    GVL.g_stTrackingQueue_B.Objects[2].Valid := TRUE;
    GVL.g_stTrackingQueue_B.Objects[2].ObjectID :=
        GVL.g_stTrackingQueue_B.NextObjectID;
    GVL.g_stTrackingQueue_B.Objects[2].ProductClassID := 1;
    GVL.g_stTrackingQueue_B.Objects[2].Reserved := FALSE;
    GVL.g_stTrackingQueue_B.Objects[2].ReservedToolID := 0;
    GVL.g_stTrackingQueue_B.Objects[2].CanPick := TRUE;
    GVL.g_stTrackingQueue_B.Objects[2].OrientationValid := TRUE;
    GVL.g_stTrackingQueue_B.Objects[2].VisionScore := 100.0;
    GVL.g_stTrackingQueue_B.Objects[2].State := E_TrackingObjectState.OBJ_READY;

    // Đặt cách Object 1 một khoảng để dễ quan sát.
    GVL.g_stTrackingQueue_B.Objects[2].VisionPos.X := 260.0;
    GVL.g_stTrackingQueue_B.Objects[2].VisionPos.Y := 0.0;
    GVL.g_stTrackingQueue_B.Objects[2].VisionPos.Z := 50.0;
    GVL.g_stTrackingQueue_B.Objects[2].VisionPos.A := 0.0;
	
	//-------------------------------------------------------------------------
	// OBJECT 2 - POSE CHUẨN TRONG HỆ CONVEYOR
	//-------------------------------------------------------------------------
	GVL.g_stTrackingQueue_B.Objects[2].PoseInConveyor.X := 260.0;
	GVL.g_stTrackingQueue_B.Objects[2].PoseInConveyor.Y := 0.0;
	GVL.g_stTrackingQueue_B.Objects[2].PoseInConveyor.Z := 50.0;
	GVL.g_stTrackingQueue_B.Objects[2].PoseInConveyor.A := 0.0;

	
	GVL.g_stTrackingQueue_B.Objects[2].CaptureConveyorPositionMM :=
		REAL_TO_LREAL(GVL.g_aConveyorRuntime[2].Status.PositionMM);

    GVL.g_stTrackingQueue_B.ValidCount := 2;
    GVL.g_stTrackingQueue_B.ActiveIndex := GVL.C_INVALID_INDEX;
	

//     GVL.g_stTrackingQueue_B.ValidCount := 1;
    GVL.g_stTrackingQueue_B.ActiveIndex := GVL.C_INVALID_INDEX;
END_IF;


//=============================================================================
// KHỞI TẠO CẤU HÌNH MẶC ĐỊNH CHO MULTI-TOOL ROBOT B
//-----------------------------------------------------------------------------
// Chỉ chạy một lần khi cấu hình chưa được khởi tạo hoặc khi người dùng yêu cầu
// khởi tạo lại. Không ghi đè cấu hình HMI trong mỗi vòng quét PLC.
//=============================================================================
IF (NOT GVL.g_xMultiToolConfigInitializedB OR GVL.g_xInitializeMultiToolConfigB) AND (1=2) THEN

    //-------------------------------------------------------------------------
    // TOOL 1
    //-------------------------------------------------------------------------
	GVL.g_aToolConfigB[1].Enable := TRUE;
	GVL.g_aToolConfigB[1].AllowTracking := TRUE;
	GVL.g_aToolConfigB[1].ToolID := 1;
	GVL.g_aToolConfigB[1].AllowedProductClassID := 0;
	

    //-------------------------------------------------------------------------
    // RECIPE 1 DÙNG CHO COMMISSIONING
    //-------------------------------------------------------------------------
    GVL.g_aMultiTrackRecipeB[1].Enable := TRUE;
    GVL.g_aMultiTrackRecipeB[1].RecipeID := 1;
    GVL.g_aMultiTrackRecipeB[1].ProductClassID := 0;
    GVL.g_aMultiTrackRecipeB[1].TargetPickCount := 1;
    GVL.g_aMultiTrackRecipeB[1].ToolEnableMask := DWORD#1;
	
	GVL.g_aToolConfigB[1].PickOffset.X := 0.0;
	GVL.g_aToolConfigB[1].PickOffset.Y := 0.0;
	GVL.g_aToolConfigB[1].PickOffset.Z := 50.0;
	GVL.g_aToolConfigB[1].PickOffset.A := 0.0;
	
	GVL.g_aToolConfigB[1].ApproachHeight := 20.0;
	GVL.g_aToolConfigB[1].UseUpDown := FALSE;
	GVL.g_aToolConfigB[1].UpDownStroke := 20.0;
	
	GVL.g_stTrackingConfig_B.RetractHeight := 20.0;
	
	
	//-------------------------------------------------------------------------
	// TOOL 2
	//-------------------------------------------------------------------------
	GVL.g_aToolConfigB[2].Enable := TRUE;
	GVL.g_aToolConfigB[2].AllowTracking := TRUE;
	GVL.g_aToolConfigB[2].ToolID := 2;
	GVL.g_aToolConfigB[2].AllowedProductClassID := 0;
	
	GVL.g_aToolConfigB[2].PickOffset.X := 0.0;
	GVL.g_aToolConfigB[2].PickOffset.Y := 0.0;
	GVL.g_aToolConfigB[2].PickOffset.Z := 50.0;
	GVL.g_aToolConfigB[2].PickOffset.A := 0.0;
	
	GVL.g_aToolConfigB[2].ApproachHeight := 20.0;
	
	// Có thể đặt khác Tool 1 để quan sát.
	GVL.g_aToolConfigB[2].UseUpDown := FALSE;
	GVL.g_aToolConfigB[2].UpDownStroke := 20.0;
	
	GVL.g_aToolConfigB[2].Priority := 2;


	//=============================================================================
	// DYNAMIC APPROACH
	//-----------------------------------------------------------------------------
	// Thông số thử nghiệm ban đầu. Có thể chỉnh lại trên HMI sau.
	//=============================================================================
	GVL.g_stTrackingConfig_B.Motion.Approach.Speed := 100.0;
	GVL.g_stTrackingConfig_B.Motion.Approach.Acceleration := 500.0;
	GVL.g_stTrackingConfig_B.Motion.Approach.Deceleration := 500.0;
	GVL.g_stTrackingConfig_B.Motion.Approach.Jerk := 1000.0;
	GVL.g_stTrackingConfig_B.Motion.Approach.BlendRadius := 0.0;
	
	GVL.g_stTrackingSimulation.VirtualEncoderStepPerCycle := -5;

    //-------------------------------------------------------------------------
    // ĐÁNH DẤU ĐÃ KHỞI TẠO
    //-------------------------------------------------------------------------
    GVL.g_xMultiToolConfigInitializedB := TRUE;
    GVL.g_xInitializeMultiToolConfigB := FALSE;

END_IF;

//=============================================================================
// PHỤC HỒI DỮ LIỆU COMMISSIONING KHI RESET MULTI-TOOL
//-----------------------------------------------------------------------------
// Chỉ dùng khi test Object cố định.
// Khi chạy Vision/Sensor thật, Object lỗi phải được loại bỏ hoặc nạp Object mới.
//=============================================================================
IF GVL.g_xMultiTrackResetTestB THEN


	//---------------------------------------------------------------------
    // RESET TOOL 1
    //---------------------------------------------------------------------
    GVL.g_aToolStatusB[1].Busy := FALSE;
    GVL.g_aToolStatusB[1].Occupied := FALSE;
    GVL.g_aToolStatusB[1].Error := FALSE;
    GVL.g_aToolStatusB[1].ErrorID := 0;
    GVL.g_aToolStatusB[1].HeldObjectID := 0;
    GVL.g_aToolStatusB[1].GripOK := FALSE;

    //---------------------------------------------------------------------
    // RESET TOOL 2
    //---------------------------------------------------------------------
    GVL.g_aToolStatusB[2].Busy := FALSE;
    GVL.g_aToolStatusB[2].Occupied := FALSE;
    GVL.g_aToolStatusB[2].Error := FALSE;
    GVL.g_aToolStatusB[2].ErrorID := 0;
    GVL.g_aToolStatusB[2].HeldObjectID := 0;
    GVL.g_aToolStatusB[2].GripOK := FALSE;
	
	// Comment lai vi dang test object thuc

//     //---------------------------------------------------------------------
//     // RESET OBJECT 1
//     //---------------------------------------------------------------------
//     GVL.g_stTrackingQueue_B.Objects[1].Valid := TRUE;
//     GVL.g_stTrackingQueue_B.Objects[1].CanPick := TRUE;
//     GVL.g_stTrackingQueue_B.Objects[1].Reserved := FALSE;
//     GVL.g_stTrackingQueue_B.Objects[1].ReservedToolID := 0;
//     GVL.g_stTrackingQueue_B.Objects[1].State :=
//         E_TrackingObjectState.OBJ_READY;
// 
//     //---------------------------------------------------------------------
//     // RESET OBJECT 2
//     //---------------------------------------------------------------------
//     GVL.g_stTrackingQueue_B.Objects[2].Valid := TRUE;
//     GVL.g_stTrackingQueue_B.Objects[2].CanPick := TRUE;
//     GVL.g_stTrackingQueue_B.Objects[2].Reserved := FALSE;
//     GVL.g_stTrackingQueue_B.Objects[2].ReservedToolID := 0;
//     GVL.g_stTrackingQueue_B.Objects[2].State :=
//         E_TrackingObjectState.OBJ_READY;
// 
//     GVL.g_stTrackingQueue_B.ValidCount := 2;
//     GVL.g_stTrackingQueue_B.ActiveIndex := GVL.C_INVALID_INDEX;

END_IF;

IF stCommandB.Reset THEN
    udiDebugCoreStartCountB := 0;
    udiDebugExecuteToCoreCountB := 0;
    udiDebugCoreRequestCountB := 0;

    xDebugCoreStartLatchedB := FALSE;
    xDebugExecuteToCoreLatchedB := FALSE;
    xDebugCoreRequestLatchedB := FALSE;
	GVL.g_xMultiTrackStartTestB := FALSE;
END_IF;

//=============================================================================
// 04. MULTI-TOOL CONTROLLER
//-----------------------------------------------------------------------------
// Controller đọc phản hồi của Core, SelectTool và ToolManager từ vòng quét trước.
//=============================================================================
fbControllerB(
    Command := stCommandB,
    CoreAccepted := fbCoreInterfaceB.Accepted,
    CoreBusy := fbCoreInterfaceB.Busy,
    CoreSyncOK := fbCoreInterfaceB.SyncOK,
    CorePCSInUse := fbCoreInterfaceB.PCSInUse,
    CoreReleased := fbCoreInterfaceB.Released,
    CoreError := fbCoreInterfaceB.Error,
    CoreErrorID := fbCoreInterfaceB.ErrorID,
    SelectToolDone := fbSelectToolB.Done,
    SelectToolError := fbSelectToolB.Error,
    SelectToolErrorID := fbSelectToolB.ErrorID,
    Queue := GVL.g_stTrackingQueue_B,
    ToolConfig := GVL.g_aToolConfigB,
    ToolStatus := GVL.g_aToolStatusB,
    Recipes := GVL.g_aMultiTrackRecipeB,
    Status := GVL.g_stMultiTrackStatusB
);


//=============================================================================
// MULTI-TOOL TRACKING RESULT LATCH
//=============================================================================

// Command mới được Controller nhận -> xóa kết quả command trước.
IF GVL.g_stMultiTrackStatusB.Accepted THEN
    GVL.g_xTrackOKB := FALSE;
    GVL.g_xTrackErrorB := FALSE;
    GVL.g_udiTrackErrorIDB := 0;
END_IF;


//-----------------------------------------------------------------------------
// TRACKING PICK HOÀN THÀNH ĐỦ SỐ LƯỢNG.
//-----------------------------------------------------------------------------
IF GVL.g_stMultiTrackStatusB.Done
AND NOT GVL.g_stMultiTrackStatusB.Error
AND GVL.g_stMultiTrackStatusB.PickedCount >= GVL.g_stMultiTrackStatusB.TargetPickCount THEN

    GVL.g_xTrackOKB := TRUE;
    GVL.g_xTrackErrorB := FALSE;
    GVL.g_udiTrackErrorIDB := 0;

    // Chốt CommandID của đúng lệnh vừa hoàn thành.
    GVL.g_udiTrackDoneCommandIDB :=
        GVL.g_stMultiTrackStatusB.ResponseCommandID;

END_IF;


//-----------------------------------------------------------------------------
// TRACKING ERROR.
//-----------------------------------------------------------------------------
IF GVL.g_stMultiTrackStatusB.Error THEN

    GVL.g_xTrackOKB := FALSE;
    GVL.g_xTrackErrorB := TRUE;
    GVL.g_udiTrackErrorIDB :=
        GVL.g_stMultiTrackStatusB.ErrorID;

END_IF;


//-----------------------------------------------------------------------------
// RESET.
//-----------------------------------------------------------------------------
IF stCommandB.Reset THEN

    GVL.g_xTrackOKB := FALSE;
    GVL.g_xTrackErrorB := FALSE;
    GVL.g_udiTrackErrorIDB := 0;
    GVL.g_udiTrackDoneCommandIDB := 0;

END_IF;



//=============================================================================
// 05. TRACKING CORE INTERFACE
//-----------------------------------------------------------------------------
// Interface giữ Execute cho Tracking Core và chỉ hạ sau khi PCS đã release.
//=============================================================================
fbCoreInterfaceB(
    Enable := TRUE,
    Reset := fbControllerB.CoreReset,
    Abort := fbControllerB.CoreAbort,
    StartTracking := fbControllerB.CoreStart,
    ReleaseTracking := fbControllerB.CoreRelease,
    ObjectIndex := fbControllerB.CoreObjectIndex,
    ToolID := fbControllerB.CoreToolID,
    PickOffset := fbControllerB.CorePickOffset,
    ApproachHeight := fbControllerB.CoreApproachHeight,
	PickSurfaceHeightMM := fbControllerB.CorePickSurfaceHeightMM,
    CoreAccepted := GVL.g_stTrackingRuntime_B.Response.Accepted,
	CoreBusy := GVL.g_stTrackingRuntime_B.Response.Busy,
	CoreSyncOK := fbTrackingManagerB.SyncOK,
	CorePCSInUse := GVL.g_stTrackingRuntime_B.PCSInfo.InUse,
	CoreReleased := fbTrackingManagerB.Released,
	CoreError := GVL.g_stTrackingRuntime_B.Response.Error,
	CoreErrorID := GVL.g_stTrackingRuntime_B.Response.ErrorID,
	UseUpDown := fbControllerB.CoreUseUpDown,
	UpDownStroke := fbControllerB.CoreUpDownStroke,
);


//=============================================================================
// 06. CHỌN TOOL/TCP ROBOT B
//-----------------------------------------------------------------------------
// FB_SelectRobotTool phải gọi SMC_GroupSetTool thực tế, không dùng placeholder.
//=============================================================================
fbSelectToolB(
    Execute := fbControllerB.SelectToolExecute,
    Reset := stCommandB.Reset,
    ToolID := fbControllerB.SelectToolID
);


// xTrackingRequestValid :=
//     fbCoreInterfaceB.ExecuteToCore
//     AND fbCoreInterfaceB.ActiveObjectIndex >= 1
//     AND fbCoreInterfaceB.ActiveObjectIndex <= GVL.C_MAX_TRACK_OBJECTS
//     AND GVL.g_stTrackingQueue_B.Objects[fbCoreInterfaceB.ActiveObjectIndex].Valid;
	
xCoreRequestValid := fbCoreInterfaceB.ExecuteToCore
AND fbCoreInterfaceB.ActiveObjectIndex >= 1
AND fbCoreInterfaceB.ActiveObjectIndex <= GVL.C_MAX_TRACK_OBJECTS
AND GVL.g_stTrackingQueue_B.Objects[fbCoreInterfaceB.ActiveObjectIndex].Valid;

rtDebugCoreStartB(CLK := fbControllerB.CoreStart);
rtDebugExecuteToCoreB(CLK := fbCoreInterfaceB.ExecuteToCore);
rtDebugCoreRequestValidB(CLK := xCoreRequestValid);

IF rtDebugCoreStartB.Q THEN
    udiDebugCoreStartCountB := udiDebugCoreStartCountB + 1;
    xDebugCoreStartLatchedB := TRUE;
END_IF;

IF rtDebugExecuteToCoreB.Q THEN
    udiDebugExecuteToCoreCountB := udiDebugExecuteToCoreCountB + 1;
    xDebugExecuteToCoreLatchedB := TRUE;
END_IF;

IF rtDebugCoreRequestValidB.Q THEN
    udiDebugCoreRequestCountB := udiDebugCoreRequestCountB + 1;
    xDebugCoreRequestLatchedB := TRUE;
END_IF;


//=============================================================================
// 07. TRACKING CORE
//-----------------------------------------------------------------------------
// Multi-tool mode luôn dùng UseExternalSelection = TRUE.
// Controller đã chọn ObjectIndex và PickOffset theo Tool.
//=============================================================================
fbTrackingManagerB(
    Execute := xCoreRequestValid,
    Reset := fbCoreInterfaceB.ResetToCore OR stCommandB.Reset,
    Config := GVL.g_stTrackingConfig_B,
    ConveyorConfig := GVL.g_aConveyorRuntime[2].Config,
    ConveyorStatus := GVL.g_aConveyorRuntime[2].Status,
    ConveyorOrigin := stConveyorOriginB,
    VacuumOK := FALSE,
    MotionAccepted := GVL.g_xTrackingMotionAcceptedB,
    MotionBusy := GVL.g_xTrackingMotionBusyB,
    MotionDone := GVL.g_xTrackingMotionDoneB,
    MotionError := GVL.g_xTrackingMotionErrorB,
    MotionErrorID := GVL.g_udiTrackingMotionErrorIDB,
    MotionAbortDone := GVL.g_xTrackingMotionAbortDoneB,
    TestFixedObjectMode := FALSE,
    FixedObjectPosition := stFixedObjectPositionB,
    UseExternalSelection := TRUE,
    ExternalObjectIndex := fbCoreInterfaceB.ActiveObjectIndex,
    ExternalPickOffset := fbCoreInterfaceB.ActivePickOffset,
    ExternalApproachHeight := fbCoreInterfaceB.ActiveApproachHeight,
    PickerSafe := fbCoreInterfaceB.PickerSafeToCore,
    Queue := GVL.g_stTrackingQueue_B,
    Runtime := GVL.g_stTrackingRuntime_B,
	ExternalUseUpDown := fbCoreInterfaceB.ActiveUseUpDown,
	ExternalUpDownStroke := fbCoreInterfaceB.ActiveUpDownStroke,
	ExternalPickSurfaceHeightMM := fbCoreInterfaceB.ActivePickSurfaceHeightMM,
);


//=============================================================================
// 08. MAP PHẢN HỒI TRACKING CORE
//-----------------------------------------------------------------------------
// Các biến này được FB_TrackingCoreInterface_A đọc ở vòng quét tiếp theo.
//=============================================================================
GVL.g_xTrackingCoreAcceptedB := GVL.g_stTrackingRuntime_B.Response.Accepted;
GVL.g_xTrackingCoreBusyB := GVL.g_stTrackingRuntime_B.Response.Busy;
GVL.g_xTrackingCoreSyncOKB := fbTrackingManagerB.SyncOK;
GVL.g_xTrackingCorePCSInUseB := GVL.g_stTrackingRuntime_B.PCSInfo.InUse;
GVL.g_xTrackingCoreReleasedB := fbTrackingManagerB.Released;
GVL.g_xTrackingCoreErrorB := GVL.g_stTrackingRuntime_B.Response.Error;
GVL.g_udiTrackingCoreErrorIDB := GVL.g_stTrackingRuntime_B.Response.ErrorID;


//=============================================================================
// 09. MOTION QUEUE ADAPTER
//-----------------------------------------------------------------------------
// Chỉ instance này được đưa motion Tracking vào Motion Queue Robot B.
//=============================================================================
fbMotionAdapterB(
    Enable := TRUE,
    Reset := fbCoreInterfaceB.ResetToCore OR stCommandB.Reset,
    Request := fbTrackingManagerB.MotionRequest,
    Abort := fbTrackingManagerB.MotionAbort,
    Target := fbTrackingManagerB.MotionTarget,
    Speed := fbTrackingManagerB.MotionSpeed,
    Acceleration := fbTrackingManagerB.MotionAcceleration,
    Deceleration := fbTrackingManagerB.MotionDeceleration,
    Jerk := fbTrackingManagerB.MotionJerk,
    BlendRadius := fbTrackingManagerB.MotionBlendRadius,
    CoordSystem := fbTrackingManagerB.MotionCoordSystem,
    Command := fbTrackingManagerB.MotionCommand,
    LogicSimulation := GVL.g_stTrackingSimulation.Mode = E_ApplicationSimulationMode.SIM_LOGIC_ONLY,
    LogicMotionDuration := GVL.g_stTrackingSimulation.LogicMotionDuration,
    Accepted => GVL.g_xTrackingMotionAcceptedB,
    Busy => GVL.g_xTrackingMotionBusyB,
    Done => GVL.g_xTrackingMotionDoneB,
    Error => GVL.g_xTrackingMotionErrorB,
    ErrorID => GVL.g_udiTrackingMotionErrorIDB,
    AbortDone => GVL.g_xTrackingMotionAbortDoneB
);


//=============================================================================
// 10. PHÂN PHỐI COMMAND TỚI TỪNG TOOL MANAGER
//-----------------------------------------------------------------------------
// Chỉ Tool có ToolID trùng Command mới nhận Execute.
// Các Tool còn lại vẫn được gọi mỗi vòng quét để duy trì Runtime và Output.
//=============================================================================
FOR uiTool := 1 TO GVL.C_MAX_TOOLS DO
	
	// Tất cả OUTPUT mặc định Active HIGH.
	GVL.g_aToolConfigB[uiTool].IO.DownDOActiveLevel := TRUE;
	GVL.g_aToolConfigB[uiTool].IO.UpDOActiveLevel := TRUE;
	GVL.g_aToolConfigB[uiTool].IO.GripDOActiveLevel := TRUE;
	GVL.g_aToolConfigB[uiTool].IO.ReleaseDOActiveLevel := TRUE;
	
	// Tất cả INPUT feedback mặc định Active HIGH.
	GVL.g_aToolConfigB[uiTool].IO.DownOKDIActiveLevel := TRUE;
	GVL.g_aToolConfigB[uiTool].IO.UpOKDIActiveLevel := TRUE;
	GVL.g_aToolConfigB[uiTool].IO.GripOKDIActiveLevel := TRUE;
	GVL.g_aToolConfigB[uiTool].IO.PartPresentDIActiveLevel := TRUE;
	
    astToolCommandB[uiTool].Execute := FALSE;
    astToolCommandB[uiTool].Reset := stCommandB.Reset;
    astToolCommandB[uiTool].Abort := stCommandB.Abort;
    astToolCommandB[uiTool].CommandID := 0;
    astToolCommandB[uiTool].ToolID := GVL.g_aToolConfigB[uiTool].ToolID;
    astToolCommandB[uiTool].CommandType := E_ToolCommandType.NONE;
    astToolCommandB[uiTool].ObjectID := 0;

    //IF fbControllerB.ToolCommand.ToolID = GVL.g_aToolConfigB[uiTool].ToolID THEN astToolCommandB[uiTool] := fbControllerB.ToolCommand; END_IF;
	
//-------------------------------------------------------------------------
	// ƯU TIÊN 1: Command từ MultiTool Tracking Controller.
	//-------------------------------------------------------------------------
	IF fbControllerB.ToolCommand.Execute
	AND fbControllerB.ToolCommand.ToolID = GVL.g_aToolConfigB[uiTool].ToolID THEN
	
		astToolCommandB[uiTool] := fbControllerB.ToolCommand;
	
	
	//-------------------------------------------------------------------------
	// ƯU TIÊN 2: Command Tool độc lập từ Interpreter.
	// Chỉ chạy khi Controller không phát Tool Command.
	//-------------------------------------------------------------------------
	ELSIF GVL.g_stInterpreterToolCommandB.Execute
	AND GVL.g_stInterpreterToolCommandB.ToolID = GVL.g_aToolConfigB[uiTool].ToolID THEN
	
		astToolCommandB[uiTool] :=
			GVL.g_stInterpreterToolCommandB;
	
	END_IF;

    fbToolManagerB[uiTool](
        Enable := GVL.g_aToolConfigB[uiTool].Enable,
        Command := astToolCommandB[uiTool],
        Config := GVL.g_aToolConfigB[uiTool],
        Status := GVL.g_aToolStatusB[uiTool]
    );
END_FOR;


//=============================================================================
// 11. BIẾN GIÁM SÁT HMI / DEBUG
//=============================================================================
GVL.g_xMultiTrackCoreExecuteB := fbCoreInterfaceB.ExecuteToCore;
GVL.g_xMultiTrackCoreResetB := fbCoreInterfaceB.ResetToCore;
GVL.g_xMultiTrackCoreAbortB := fbCoreInterfaceB.AbortToCore;
GVL.g_xMultiTrackPickerSafeB := fbCoreInterfaceB.PickerSafeToCore;
GVL.g_uiMultiTrackObjectIndexB := fbCoreInterfaceB.ActiveObjectIndex;
GVL.g_uiMultiTrackToolIDB := fbCoreInterfaceB.ActiveToolID;
GVL.g_stMultiTrackPickOffsetB := fbCoreInterfaceB.ActivePickOffset;
GVL.g_rMultiTrackApproachHeightB := fbCoreInterfaceB.ActiveApproachHeight;
GVL.g_xSelectToolExecuteB := fbControllerB.SelectToolExecute;
GVL.g_uiSelectToolIDB := fbControllerB.SelectToolID;
GVL.g_stSelectToolTCPB := fbControllerB.SelectToolTCP;
GVL.g_xSelectToolDoneB := fbSelectToolB.Done;
GVL.g_xSelectToolErrorB := fbSelectToolB.Error;
GVL.g_udiSelectToolErrorIDB := fbSelectToolB.ErrorID;


//=============================================================================
// 12. OUTPUT CŨ CỦA TRACKING CORE
//-----------------------------------------------------------------------------
// Multi-tool mode không dùng VacuumCommand/BlowCommand; giữ map để debug.
//=============================================================================
GVL.g_xTrackingVacuumOutputB := fbTrackingManagerB.VacuumCommand;
GVL.g_xTrackingBlowOutputB := fbTrackingManagerB.BlowCommand;

END_PROGRAM

// Just_Motion_Control_x86_64_Linux_SM_WV/Application/FB_/ConveyorTrack/FB_MultiToolTrackingController_B
FUNCTION_BLOCK FB_MultiToolTrackingController_B
VAR_INPUT
    Command : ST_MultiToolTrackingCommand; // Biến nội bộ Command.
    CoreAccepted : BOOL; // Biến nội bộ CoreAccepted.
    CoreBusy : BOOL; // Biến nội bộ CoreBusy.
    CoreSyncOK : BOOL; // Biến nội bộ CoreSyncOK.
    CorePCSInUse : BOOL; // Biến nội bộ CorePCSInUse.
    CoreReleased : BOOL; // Biến nội bộ CoreReleased.
    CoreError : BOOL; // Biến nội bộ CoreError.
    CoreErrorID : UDINT; // Biến nội bộ CoreErrorID.
    SelectToolDone : BOOL; // Biến nội bộ SelectToolDone.
    SelectToolError : BOOL; // Biến nội bộ SelectToolError.
    SelectToolErrorID : UDINT; // Biến nội bộ SelectToolErrorID.
END_VAR

VAR_IN_OUT
    Queue : ST_TRACKING_QUEUE; // Biến nội bộ Queue.
    ToolConfig : ARRAY[0..GVL.C_MAX_TOOLS] OF ST_ToolConfig; // Biến nội bộ ToolConfig.
    ToolStatus : ARRAY[0..GVL.C_MAX_TOOLS] OF ST_ToolStatus; // Biến nội bộ ToolStatus.
    Recipes : ARRAY[0..GVL.C_MAX_TRACK_RECIPES] OF ST_MultiToolTrackingRecipe; // Biến nội bộ Recipes.
    Status : ST_MultiToolTrackingStatus; // Biến nội bộ Status.
END_VAR

VAR_OUTPUT
    CoreStart : BOOL; // Biến nội bộ CoreStart.
    CoreRelease : BOOL; // Biến nội bộ CoreRelease.
    CoreAbort : BOOL; // Biến nội bộ CoreAbort.
    CoreReset : BOOL; // Biến nội bộ CoreReset.
    CoreObjectIndex : UINT; // Biến nội bộ CoreObjectIndex.
    CoreToolID : UINT; // Biến nội bộ CoreToolID.
    CorePickOffset : ST_POS; // Biến nội bộ CorePickOffset.
    CoreApproachHeight : REAL; // Biến nội bộ CoreApproachHeight.
    ToolCommand : ST_ToolCommand; // Biến nội bộ ToolCommand.
    SelectToolExecute : BOOL; // Biến nội bộ SelectToolExecute.
    SelectToolID : UINT; // Biến nội bộ SelectToolID.
    SelectToolTCP : ST_POS; // Biến nội bộ SelectToolTCP.
    CoreUseUpDown : BOOL; // Biến nội bộ CoreUseUpDown.
    CoreUpDownStroke : REAL; // Biến nội bộ CoreUpDownStroke.
    CorePickSurfaceHeightMM : REAL; // Biến nội bộ CorePickSurfaceHeightMM.
END_VAR

VAR
    rtExecute : R_TRIG; // Biến nội bộ rtExecute.
    fbScheduler : FB_ToolObjectScheduler; // Biến nội bộ fbScheduler.
    stRecipe : ST_MultiToolTrackingRecipe; // Biến nội bộ stRecipe.
    uiToolIndex : UINT; // Biến nội bộ uiToolIndex.
    uiObjectIndex : UINT; // Biến nội bộ uiObjectIndex.
    uiTargetCount : UINT; // Biến nội bộ uiTargetCount.
    dwToolMask : DWORD; // Biến nội bộ dwToolMask.
    udiToolCommandID : UDINT; // Biến nội bộ udiToolCommandID.
    xCommandIssued : BOOL; // Biến nội bộ xCommandIssued.
    xReleaseArmed : BOOL; // TRUE sau khi Controller đã giữ CoreRelease ít nhất một vòng quét. Ngăn CoreReleased cũ làm bỏ qua tín hiệu PickerSafe.
    udiLastAcceptedCommandID : UDINT := 0; // Biến nội bộ udiLastAcceptedCommandID.
END_VAR

(*
===============================================================================
FB_MultiToolTrackingController_A

MỤC ĐÍCH
    Điều phối một lệnh TRACK_ON cho Robot B.

CHU TRÌNH
    IDLE
    -> LOAD_RECIPE
    -> SELECT_ASSIGNMENT
    -> SELECT_TOOL
    -> START_TRACKING
    -> WAIT_SYNC
    -> TOOL_DOWN
    -> TOOL_GRIP
    -> TOOL_UP
    -> RELEASE_TRACKING
    -> STORE_RESULT
    -> lặp đến khi đủ TargetPickCount
    -> COMPLETE

TRÁCH NHIỆM
    - Không gọi Motion trực tiếp.
    - Không gọi MC_TrackConveyorBelt trực tiếp.
    - Không ghi IO trực tiếp.
    - Chỉ điều phối Tracking Core, Tool Manager và Select Tool.
===============================================================================
*)
//=============================================================================
// DEFAULT PULSE OUTPUTS
//=============================================================================
Status.Accepted := FALSE;
Status.Done := FALSE;
CoreStart := FALSE;
CoreRelease := FALSE;
CoreAbort := FALSE;
CoreReset := FALSE;
ToolCommand.Execute := FALSE;
SelectToolExecute := FALSE;

//=============================================================================
// RESET
//=============================================================================
IF Command.Reset THEN
    Status.State := E_MultiTrackState.IDLE;
    Status.Busy := FALSE;
    Status.Error := FALSE;
    Status.ErrorID := 0;
    Status.PickedCount := 0;
    Status.SelectedToolID := 0;
    Status.SelectedObjectID := 0;
    CoreReset := TRUE;
    xCommandIssued := FALSE;
	xReleaseArmed := FALSE;
	udiLastAcceptedCommandID := 0;
    RETURN;
END_IF;

//=============================================================================
// ABORT
//=============================================================================
IF Command.Abort THEN 
	Status.State := E_MultiTrackState.ABORTING; 
	xReleaseArmed := FALSE;
END_IF;

// //=============================================================================
// // START COMMAND
// //=============================================================================
// rtExecute(CLK := Command.Execute);
// 
// IF rtExecute.Q AND Status.State = E_MultiTrackState.IDLE THEN
//     Status.Accepted := TRUE;
//     Status.Busy := TRUE;
//     Status.Error := FALSE;
//     Status.ErrorID := 0;
//     Status.ResponseCommandID := Command.CommandID;
//     Status.PickedCount := 0;
//     Status.OccupiedToolMask := 0;
//     Status.State := E_MultiTrackState.LOAD_RECIPE;
// END_IF;

//=============================================================================
// START NEW COMMAND
//-----------------------------------------------------------------------------
// Không phụ thuộc riêng cạnh Execute.
// CommandID là khóa transaction chính.
//=============================================================================
IF Command.Execute
AND Command.CommandID <> 0
AND Command.CommandID <> udiLastAcceptedCommandID
AND Status.State = E_MultiTrackState.IDLE THEN

    udiLastAcceptedCommandID := Command.CommandID;

    Status.Accepted := TRUE;
    Status.Busy := TRUE;
    Status.Error := FALSE;
    Status.ErrorID := 0;

    Status.ResponseCommandID := Command.CommandID;
    Status.PickedCount := 0;
    Status.OccupiedToolMask := 0;

    Status.State := E_MultiTrackState.LOAD_RECIPE;

END_IF;


//=============================================================================
// STATE MACHINE
//=============================================================================
CASE Status.State OF

    E_MultiTrackState.IDLE:
        Status.Busy := FALSE;

    //-------------------------------------------------------------------------
    // Đọc Recipe và áp dụng tham số Override từ Interpreter.
    //-------------------------------------------------------------------------
    E_MultiTrackState.LOAD_RECIPE:
        IF Command.RecipeID = 0 OR Command.RecipeID > 32 OR NOT Recipes[Command.RecipeID].Enable THEN
            Status.Error := TRUE;
            Status.ErrorID := 9401;
            Status.State := E_MultiTrackState.ERROR;
        ELSE
            stRecipe := Recipes[Command.RecipeID];
            Status.ActiveRecipeID := stRecipe.RecipeID;
            IF Command.TargetPickCountOverride > 0 THEN uiTargetCount := Command.TargetPickCountOverride; ELSE uiTargetCount := stRecipe.TargetPickCount; END_IF;
            IF Command.ToolMaskOverride <> 0 THEN dwToolMask := Command.ToolMaskOverride; ELSE dwToolMask := stRecipe.ToolEnableMask; END_IF;
            Status.TargetPickCount := uiTargetCount;
            Status.State := E_MultiTrackState.VALIDATE_TOOLS;
        END_IF;

    //-------------------------------------------------------------------------
    // Kiểm tra nhanh cấu hình trước khi chạy.
    //-------------------------------------------------------------------------
    E_MultiTrackState.VALIDATE_TOOLS:
        IF uiTargetCount = 0 OR dwToolMask = 0 THEN
            Status.Error := TRUE;
            Status.ErrorID := 9402;
            Status.State := E_MultiTrackState.ERROR;
        ELSE
            Status.State := E_MultiTrackState.SELECT_ASSIGNMENT;
        END_IF;

    //-------------------------------------------------------------------------
    // Tìm một Tool rảnh và một Object phù hợp.
    //-------------------------------------------------------------------------
    E_MultiTrackState.SELECT_ASSIGNMENT:

		fbScheduler(
			Execute := TRUE,
			Recipe := stRecipe,
			ToolMask := dwToolMask,
			Queue := Queue,
			ToolConfig := ToolConfig,
			ToolStatus := ToolStatus
		);
	
		IF fbScheduler.Done AND fbScheduler.Valid THEN
			uiToolIndex := fbScheduler.ToolIndex;
			uiObjectIndex := fbScheduler.ObjectIndex;
	
			// Controller chỉ ghi Tool được phân công.
			// Tracking Manager là khối duy nhất được Reserve Object.
			Queue.Objects[uiObjectIndex].ReservedToolID := ToolConfig[uiToolIndex].ToolID;
	
			Status.SelectedToolID := ToolConfig[uiToolIndex].ToolID;
			Status.SelectedObjectID := Queue.Objects[uiObjectIndex].ObjectID;
	
			xCommandIssued := FALSE;
			Status.State := E_MultiTrackState.SELECT_ROBOT_TOOL;
		END_IF;

		
	//-------------------------------------------------------------------------
	// Chọn TCP/Tool cho Robot B.
	//-------------------------------------------------------------------------
	E_MultiTrackState.SELECT_ROBOT_TOOL:
	
		SelectToolID := ToolConfig[uiToolIndex].ToolID;
		SelectToolTCP := ToolConfig[uiToolIndex].ToolTCP;
		SelectToolExecute := TRUE;
	
		IF SelectToolDone THEN
			SelectToolExecute := FALSE;
			xCommandIssued := FALSE;
			Status.State := E_MultiTrackState.START_TRACKING;
	
		ELSIF SelectToolError THEN
			SelectToolExecute := FALSE;
			Status.Error := TRUE;
			Status.ErrorID := SelectToolErrorID;
			Status.State := E_MultiTrackState.ERROR;
		END_IF;
	
	
    //-------------------------------------------------------------------------
    // Phát request tới Tracking Core.
    //-------------------------------------------------------------------------
    E_MultiTrackState.START_TRACKING:
        CoreObjectIndex := uiObjectIndex;
        CoreToolID := ToolConfig[uiToolIndex].ToolID;
        CorePickOffset := ToolConfig[uiToolIndex].PickOffset;
        CoreApproachHeight := ToolConfig[uiToolIndex].ApproachHeight;
		CorePickSurfaceHeightMM := stRecipe.PickSurfaceHeightMM;
        CoreUseUpDown := ToolConfig[uiToolIndex].UseUpDown;
        CoreUpDownStroke := ToolConfig[uiToolIndex].UpDownStroke;
        CoreStart := TRUE;

        IF CoreAccepted OR CoreBusy THEN
            Queue.Objects[uiObjectIndex].State := E_TrackingObjectState.OBJ_TRACKING;
            Status.State := E_MultiTrackState.WAIT_SYNC;

        ELSIF CoreError THEN
            Status.Error := TRUE;
            Status.ErrorID := CoreErrorID;
            Status.State := E_MultiTrackState.ERROR;
        END_IF;

    //-------------------------------------------------------------------------
    // Chờ Robot tới Approach trong PCS và PCS vẫn InUse.
    //-------------------------------------------------------------------------
    E_MultiTrackState.WAIT_SYNC:
        Status.TrackingSyncOK := CoreSyncOK;
        Status.PCSInUse := CorePCSInUse;

        IF CoreSyncOK AND CorePCSInUse THEN
            xCommandIssued := FALSE;

            IF ToolConfig[uiToolIndex].UseUpDown THEN
                Status.State := E_MultiTrackState.TOOL_DOWN;
            ELSE
                Status.State := E_MultiTrackState.TOOL_GRIP;
            END_IF;

        ELSIF CoreError THEN
            Status.Error := TRUE;
            Status.ErrorID := CoreErrorID;
            Status.State := E_MultiTrackState.ERROR;
        END_IF;


    //-------------------------------------------------------------------------
	// COMMAND TOOL DOWN
	//-------------------------------------------------------------------------
	E_MultiTrackState.TOOL_DOWN:
	
		udiToolCommandID := udiToolCommandID + 1;
	
		ToolCommand.CommandID := udiToolCommandID;
		ToolCommand.ToolID := ToolConfig[uiToolIndex].ToolID;
		ToolCommand.CommandType := E_ToolCommandType.DOWN;
		ToolCommand.ObjectID := Queue.Objects[uiObjectIndex].ObjectID;
		ToolCommand.Execute := TRUE;
	
		Status.State := E_MultiTrackState.WAIT_TOOL_DOWN;
	
	
	//-------------------------------------------------------------------------
	// WAIT TOOL DOWN
	//-------------------------------------------------------------------------
	E_MultiTrackState.WAIT_TOOL_DOWN:
	
		IF ToolStatus[uiToolIndex].Done
		AND ToolStatus[uiToolIndex].ResponseCommandID = udiToolCommandID THEN
	
			Status.State := E_MultiTrackState.TOOL_GRIP;
	
		ELSIF ToolStatus[uiToolIndex].Error THEN
	
			Status.Error := TRUE;
			Status.ErrorID := ToolStatus[uiToolIndex].ErrorID;
			Status.State := E_MultiTrackState.ERROR;
	
		END_IF;
	
	
	//-------------------------------------------------------------------------
	// COMMAND TOOL GRIP
	//-------------------------------------------------------------------------
	E_MultiTrackState.TOOL_GRIP:
	
		udiToolCommandID := udiToolCommandID + 1;
	
		ToolCommand.CommandID := udiToolCommandID;
		ToolCommand.ToolID := ToolConfig[uiToolIndex].ToolID;
		ToolCommand.CommandType := E_ToolCommandType.GRIP;
		ToolCommand.ObjectID := Queue.Objects[uiObjectIndex].ObjectID;
		ToolCommand.Execute := TRUE;
	
		Status.State := E_MultiTrackState.WAIT_TOOL_GRIP;
	
	
	//-------------------------------------------------------------------------
	// WAIT TOOL GRIP
	//-------------------------------------------------------------------------
	E_MultiTrackState.WAIT_TOOL_GRIP:
	
		 IF ToolStatus[uiToolIndex].Done
        AND ToolStatus[uiToolIndex].ResponseCommandID = udiToolCommandID THEN

            IF ToolConfig[uiToolIndex].UseUpDown THEN
                Status.State := E_MultiTrackState.TOOL_UP;
            ELSE
                Status.State := E_MultiTrackState.RELEASE_TRACKING;
            END_IF;

        ELSIF ToolStatus[uiToolIndex].Error THEN
            Status.Error := TRUE;
            Status.ErrorID := ToolStatus[uiToolIndex].ErrorID;
            Status.State := E_MultiTrackState.ERROR;
        END_IF;
	
	
	//-------------------------------------------------------------------------
	// COMMAND TOOL UP
	//-------------------------------------------------------------------------
	E_MultiTrackState.TOOL_UP:
	
		udiToolCommandID := udiToolCommandID + 1;
	
		ToolCommand.CommandID := udiToolCommandID;
		ToolCommand.ToolID := ToolConfig[uiToolIndex].ToolID;
		ToolCommand.CommandType := E_ToolCommandType.UP;
		ToolCommand.ObjectID := Queue.Objects[uiObjectIndex].ObjectID;
		ToolCommand.Execute := TRUE;
	
		Status.State := E_MultiTrackState.WAIT_TOOL_UP;
	
	
	//-------------------------------------------------------------------------
	// WAIT TOOL UP
	//-------------------------------------------------------------------------
	E_MultiTrackState.WAIT_TOOL_UP:
	
		IF ToolStatus[uiToolIndex].Done
			AND ToolStatus[uiToolIndex].ResponseCommandID = udiToolCommandID THEN
		
				// Chuẩn bị một chu trình Release mới.
				xReleaseArmed := FALSE;
		
				Status.State := E_MultiTrackState.RELEASE_TRACKING;
		
			ELSIF ToolStatus[uiToolIndex].Error THEN
		
				Status.Error := TRUE;
				Status.ErrorID := ToolStatus[uiToolIndex].ErrorID;
				Status.State := E_MultiTrackState.ERROR;
		
			END_IF;

    //-------------------------------------------------------------------------
	// Báo PickerSafe để Tracking Core chạy Exit/Release PCS.
	//-------------------------------------------------------------------------
	E_MultiTrackState.RELEASE_TRACKING:
	
		// Phải giữ TRUE liên tục để Core Interface nhận được yêu cầu.
		CoreRelease := TRUE;
	
		// Vòng quét đầu tiên chỉ phát yêu cầu Release.
		// Không kiểm tra CoreReleased trong cùng vòng quét này.
		IF NOT xReleaseArmed THEN
	
			xReleaseArmed := TRUE;
	
		ELSE
	
			// Chỉ chấp nhận Released sau khi CoreRelease
			// đã được giữ ít nhất một vòng quét.
			IF CoreReleased THEN
	
				xReleaseArmed := FALSE;
				Status.State := E_MultiTrackState.STORE_RESULT;
	
			ELSIF CoreError THEN
	
				xReleaseArmed := FALSE;
				Status.Error := TRUE;
				Status.ErrorID := CoreErrorID;
				Status.State := E_MultiTrackState.ERROR;
				xReleaseArmed := FALSE;
			END_IF;
	
		END_IF;

    //-------------------------------------------------------------------------
    // Lưu kết quả Pick của Tool hiện tại.
    //-------------------------------------------------------------------------
    E_MultiTrackState.STORE_RESULT:
        Queue.Objects[uiObjectIndex].Reserved := FALSE;
        Queue.Objects[uiObjectIndex].State := E_TrackingObjectState.OBJ_PICKED;
        Status.PickedCount := Status.PickedCount + 1;
        Status.OccupiedToolMask := Status.OccupiedToolMask OR SHL(DWORD#1, uiToolIndex - 1);
        Status.State := E_MultiTrackState.CHECK_COUNT;

    //-------------------------------------------------------------------------
    // Đủ số lượng thì Done; chưa đủ thì chọn Tool/Object tiếp theo.
    //-------------------------------------------------------------------------
    E_MultiTrackState.CHECK_COUNT:
        IF Status.PickedCount >= uiTargetCount THEN
            Status.State := E_MultiTrackState.COMPLETE;
        ELSE
            Status.SelectedToolID := 0;
            Status.SelectedObjectID := 0;
            Status.TrackingSyncOK := FALSE;
            Status.PCSInUse := FALSE;
            Status.State := E_MultiTrackState.SELECT_ASSIGNMENT;
        END_IF;

    E_MultiTrackState.COMPLETE:
        Status.Busy := FALSE;
        Status.Done := TRUE;
        IF NOT Command.Execute THEN Status.State := E_MultiTrackState.IDLE; END_IF;

    E_MultiTrackState.ABORTING:
        CoreAbort := TRUE;
        Status.Busy := FALSE;
        Status.Error := TRUE;
        Status.ErrorID := 9499;
        Status.State := E_MultiTrackState.ERROR;

    E_MultiTrackState.ERROR:
        Status.Busy := FALSE;
        Status.Error := TRUE;
        IF NOT Command.Execute THEN Status.State := E_MultiTrackState.IDLE; END_IF;

END_CASE;

END_FUNCTION_BLOCK

// Just_Motion_Control_x86_64_Linux_SM_WV/Application/FB_/ConveyorTrack/FB_TrackingCoreInterface_B
FUNCTION_BLOCK FB_TrackingCoreInterface_B
VAR_INPUT
    Enable : BOOL; // Biến nội bộ Enable.
    Reset : BOOL; // Biến nội bộ Reset.
    Abort : BOOL; // Biến nội bộ Abort.
    StartTracking : BOOL; // Biến nội bộ StartTracking.
    ReleaseTracking : BOOL; // Biến nội bộ ReleaseTracking.
    ObjectIndex : UINT; // Biến nội bộ ObjectIndex.
    ToolID : UINT; // Biến nội bộ ToolID.
    PickOffset : ST_POS; // Biến nội bộ PickOffset.
    ApproachHeight : REAL; // Biến nội bộ ApproachHeight.
    PickSurfaceHeightMM : REAL; // Biến nội bộ PickSurfaceHeightMM.
    CoreAccepted : BOOL; // Biến nội bộ CoreAccepted.
    CoreBusy : BOOL; // Biến nội bộ CoreBusy.
    CoreSyncOK : BOOL; // Biến nội bộ CoreSyncOK.
    CorePCSInUse : BOOL; // Biến nội bộ CorePCSInUse.
    CoreReleased : BOOL; // Biến nội bộ CoreReleased.
    CoreError : BOOL; // Biến nội bộ CoreError.
    CoreErrorID : UDINT; // Biến nội bộ CoreErrorID.
    UseUpDown : BOOL; // Biến nội bộ UseUpDown.
    UpDownStroke : REAL; // Biến nội bộ UpDownStroke.
END_VAR

VAR_OUTPUT
    ExecuteToCore : BOOL; // Biến nội bộ ExecuteToCore.
    ResetToCore : BOOL; // Biến nội bộ ResetToCore.
    AbortToCore : BOOL; // Biến nội bộ AbortToCore.
    PickerSafeToCore : BOOL; // Biến nội bộ PickerSafeToCore.
    ActiveObjectIndex : UINT; // Biến nội bộ ActiveObjectIndex.
    ActiveToolID : UINT; // Biến nội bộ ActiveToolID.
    ActivePickOffset : ST_POS; // Biến nội bộ ActivePickOffset.
    ActiveApproachHeight : REAL; // Biến nội bộ ActiveApproachHeight.
    ActivePickSurfaceHeightMM : REAL; // Biến nội bộ ActivePickSurfaceHeightMM.
    Accepted : BOOL; // Biến nội bộ Accepted.
    Busy : BOOL; // Biến nội bộ Busy.
    SyncOK : BOOL; // Biến nội bộ SyncOK.
    PCSInUse : BOOL; // Biến nội bộ PCSInUse.
    Released : BOOL; // Biến nội bộ Released.
    Error : BOOL; // Biến nội bộ Error.
    ErrorID : UDINT; // Biến nội bộ ErrorID.
    ActiveUseUpDown : BOOL; // Biến nội bộ ActiveUseUpDown.
    ActiveUpDownStroke : REAL; // Biến nội bộ ActiveUpDownStroke.
END_VAR

VAR
    rtStart : R_TRIG; // Biến nội bộ rtStart.
    xRequestLatched : BOOL := FALSE; // Biến nội bộ xRequestLatched.
    xReleaseRequested : BOOL := FALSE; // TRUE sau khi Controller yêu cầu kết thúc Tracking.
    rtCoreReleased : R_TRIG; // Bắt cạnh lên của tín hiệu CoreReleased.
    xCoreWasBusy : BOOL := FALSE; // Biến nội bộ xCoreWasBusy.
    xCoreWasInUse : BOOL := FALSE; // Biến nội bộ xCoreWasInUse.
END_VAR

(*
===============================================================================
FB_TrackingCoreInterface_A

MỤC ĐÍCH
    Chuẩn hóa handshake giữa MultiTool Controller và
    FB_CONVEYOR_TRACKING_MANAGER.
===============================================================================
*)

//=============================================================================
// BẮT CẠNH TÍN HIỆU
//=============================================================================
rtStart(CLK := StartTracking);
rtCoreReleased(CLK := CoreReleased);


//=============================================================================
// OUTPUT MẶC ĐỊNH MỖI VÒNG QUÉT
//=============================================================================
ResetToCore := FALSE;
AbortToCore := FALSE;
Released := FALSE;

Accepted := CoreAccepted AND xRequestLatched;
Busy := CoreBusy AND xRequestLatched;
SyncOK := CoreSyncOK AND xRequestLatched;
PCSInUse := CorePCSInUse AND xRequestLatched;
Error := CoreError AND xRequestLatched;


IF Error THEN
    ErrorID := CoreErrorID;
ELSE
    ErrorID := 0;
END_IF;


//=============================================================================
// RESET / DISABLE
//=============================================================================
IF Reset OR NOT Enable THEN
    ExecuteToCore := FALSE;
    ResetToCore := Reset;
    AbortToCore := FALSE;
    PickerSafeToCore := FALSE;
    Released := FALSE;

    xRequestLatched := FALSE;
    xReleaseRequested := FALSE;
    xCoreWasBusy := FALSE;
    xCoreWasInUse := FALSE;

    ActiveObjectIndex := 0;
    ActiveToolID := 0;
    ActivePickOffset.X := 0.0;
    ActivePickOffset.Y := 0.0;
    ActivePickOffset.Z := 0.0;
    ActivePickOffset.A := 0.0;
    ActiveApproachHeight := 0.0;

    Accepted := FALSE;
    Busy := FALSE;
    SyncOK := FALSE;
    PCSInUse := FALSE;
    Error := FALSE;
    ErrorID := 0;
	ActiveUseUpDown := FALSE;
	ActiveUpDownStroke := 0.0;
	ActivePickSurfaceHeightMM := 0.0;

    RETURN;
END_IF;


//=============================================================================
// ABORT
//=============================================================================
IF Abort THEN
    ExecuteToCore := FALSE;
    ResetToCore := FALSE;
    AbortToCore := TRUE;
    PickerSafeToCore := FALSE;
    Released := FALSE;

    xRequestLatched := FALSE;
    xReleaseRequested := FALSE;
    xCoreWasBusy := FALSE;
    xCoreWasInUse := FALSE;

    Accepted := FALSE;
    Busy := FALSE;
    SyncOK := FALSE;
    PCSInUse := FALSE;
	
	ActiveUseUpDown := FALSE;
	ActiveUpDownStroke := 0.0;
    RETURN;
END_IF;


//=============================================================================
// START TRACKING REQUEST
//=============================================================================
IF rtStart.Q AND NOT xRequestLatched THEN
    IF ObjectIndex >= 1
    AND ObjectIndex <= GVL.C_MAX_TRACK_OBJECTS THEN

        ActiveObjectIndex := ObjectIndex;
        ActiveToolID := ToolID;
        ActivePickOffset := PickOffset;
        ActiveApproachHeight := ApproachHeight;
		ActivePickSurfaceHeightMM := PickSurfaceHeightMM;
        ActiveUseUpDown := UseUpDown;
        ActiveUpDownStroke := UpDownStroke;

        xRequestLatched := TRUE;
        xReleaseRequested := FALSE;
    END_IF;

END_IF;


//=============================================================================
// GIỮ EXECUTE TRONG TOÀN BỘ REQUEST
//=============================================================================
ExecuteToCore := xRequestLatched;

// Nhận yêu cầu release từ Controller.
IF ReleaseTracking AND xRequestLatched THEN
    xReleaseRequested := TRUE;
END_IF;

PickerSafeToCore := xRequestLatched AND xReleaseRequested;

// Chỉ đóng request khi Manager đã phát Released.
IF rtCoreReleased.Q
AND xRequestLatched
AND xReleaseRequested THEN
    Released := TRUE;
    ExecuteToCore := FALSE;
    PickerSafeToCore := FALSE;

    xRequestLatched := FALSE;
    xReleaseRequested := FALSE;

    ActiveObjectIndex := 0;
    ActiveToolID := 0;
	
	ActiveUseUpDown := FALSE;
	ActiveUpDownStroke := 0.0;
	
END_IF;

END_FUNCTION_BLOCK

// Just_Motion_Control_x86_64_Linux_SM_WV/Application/FB_/ConveyorTrack/FB_CONVEYOR_TRACKING_MANAGER_B
FUNCTION_BLOCK FB_CONVEYOR_TRACKING_MANAGER_B
VAR_INPUT
    Execute : BOOL; // Biến nội bộ Execute.
    Reset : BOOL; // Biến nội bộ Reset.
    Config : ST_TRACKING_CONFIG; // Biến nội bộ Config.
    ConveyorConfig : ST_CONVEYOR_CONFIG; // Biến nội bộ ConveyorConfig.
    ConveyorStatus : ST_CONVEYOR_STATUS; // Biến nội bộ ConveyorStatus.
    ConveyorOrigin : MC_COORD_REF; // Biến nội bộ ConveyorOrigin.
    VacuumOK : BOOL; // Biến nội bộ VacuumOK.
    MotionAccepted : BOOL; // Biến nội bộ MotionAccepted.
    MotionBusy : BOOL; // Biến nội bộ MotionBusy.
    MotionDone : BOOL; // Biến nội bộ MotionDone.
    MotionError : BOOL; // Biến nội bộ MotionError.
    MotionErrorID : UDINT; // Biến nội bộ MotionErrorID.
    MotionAbortDone : BOOL; // Biến nội bộ MotionAbortDone.
    TestFixedObjectMode : BOOL; // Biến nội bộ TestFixedObjectMode.
    FixedObjectPosition : MC_COORD_REF; // Biến nội bộ FixedObjectPosition.
    UseExternalSelection : BOOL; // Multi-tool external control.
    ExternalObjectIndex : UINT; // Biến nội bộ ExternalObjectIndex.
    ExternalPickOffset : ST_POS; // Biến nội bộ ExternalPickOffset.
    ExternalApproachHeight : REAL; // Biến nội bộ ExternalApproachHeight.
    PickerSafe : BOOL; // Biến nội bộ PickerSafe.
    ExternalUseUpDown : BOOL; // Biến nội bộ ExternalUseUpDown.
    ExternalUpDownStroke : REAL; // Biến nội bộ ExternalUpDownStroke.
    ExternalPickSurfaceHeightMM : REAL; // Chiều cao mặt cần hút của sản phẩm. Được lấy từ Recipe khi chạy MultiTool.
END_VAR

VAR_OUTPUT
    VacuumCommand : BOOL; // Biến nội bộ VacuumCommand.
    BlowCommand : BOOL; // Biến nội bộ BlowCommand.
    TrackingActive : BOOL; // Biến nội bộ TrackingActive.
    MotionRequest : BOOL; // Biến nội bộ MotionRequest.
    MotionAbort : BOOL; // Biến nội bộ MotionAbort.
    MotionTarget : ST_POS; // Biến nội bộ MotionTarget.
    MotionSpeed : REAL; // Biến nội bộ MotionSpeed.
    MotionAcceleration : REAL; // Biến nội bộ MotionAcceleration.
    MotionDeceleration : REAL; // Biến nội bộ MotionDeceleration.
    MotionJerk : REAL; // Biến nội bộ MotionJerk.
    MotionBlendRadius : REAL; // Biến nội bộ MotionBlendRadius.
    MotionCoordSystem : E_AppCoordSystem; // Biến nội bộ MotionCoordSystem.
    MotionCommand : UINT; // Biến nội bộ MotionCommand.
    SyncOK : BOOL; // Multi-tool handshake.
    Released : BOOL; // Biến nội bộ Released.
END_VAR

VAR_IN_OUT
    Queue : ST_TRACKING_QUEUE; // Biến nội bộ Queue.
    Runtime : ST_TRACKING_RUNTIME; // Biến nội bộ Runtime.
END_VAR

VAR
    fbTrackBelt : MC_TrackConveyorBelt; // Biến nội bộ fbTrackBelt.
    xTrackExecute : BOOL; // Biến nội bộ xTrackExecute.
    uiSelectedIndex : UINT; // Biến nội bộ uiSelectedIndex.
    stSelectedObject : ST_TRACKING_OBJECT; // Biến nội bộ stSelectedObject.
    xMotionIssued : BOOL; // Biến nội bộ xMotionIssued.
    xMotionRequestPending : BOOL; // Biến nội bộ xMotionRequestPending.
    xMotionActive : BOOL; // Biến nội bộ xMotionActive.
    xVacuumCaptured : BOOL; // Biến nội bộ xVacuumCaptured.
    tonPickDelay : TON; // Biến nội bộ tonPickDelay.
    tonVacuumTimeout : TON; // Biến nội bộ tonVacuumTimeout.
    tonBlow : TON; // Biến nội bộ tonBlow.
    stConveyorOriginSMC : MC_COORD_REF; // Biến nội bộ stConveyorOriginSMC.
    stInitialObjectSMC : MC_COORD_REF; // Biến nội bộ stInitialObjectSMC.
    stExitPCSTarget : ST_POS; // Biến nội bộ stExitPCSTarget.
    xExitPCSTargetValid : BOOL := FALSE; // Biến nội bộ xExitPCSTargetValid.
    rExitPCSOffsetZ : REAL := 5.0; // Biến nội bộ rExitPCSOffsetZ.
    rExitPCSOffsetX : REAL := 15.0; // Biến nội bộ rExitPCSOffsetX.
    rExitPCSMaxZ : REAL := 320.0; // Biến nội bộ rExitPCSMaxZ.
    stToolSyncPos : ST_POS; // Biến nội bộ stToolSyncPos.
    xPickPositionReady : BOOL; // Biến nội bộ xPickPositionReady.
    xPickerSafeArmed : BOOL; // Biến nội bộ xPickerSafeArmed.
    xMotionDoneArmed : BOOL; // Biến nội bộ xMotionDoneArmed.
    xPickMotionBusySeen : BOOL; // xác nhận lệnh xuống Pick thực sự chạy.
    xRetractMotionBusySeen : BOOL; // xác nhận lệnh nâng Retract thực sự chạy.
    lrConveyorDeltaAtPCS : LREAL; // Biến nội bộ lrConveyorDeltaAtPCS.
    xPCSStartCaptured : BOOL; // TRUE khi đã chụp vị trí Conveyor cho lần tạo PCS hiện tại.
    lrConveyorPosAtPCSStart : LREAL; // Vị trí Conveyor tại thời điểm chuẩn bị phát cạnh Track Execute.
    lrDeltaCaptureToPCS : LREAL; // Conveyor đã dịch từ lúc Object được Sensor/Vision Capture tới lúc tạo PCS.
END_VAR

(*
===============================================================================
FB_CONVEYOR_TRACKING_MANAGER - MULTI-TOOL CORE V2
===============================================================================
- Giữ chế độ Tracking Pick cũ khi UseExternalSelection = FALSE.
- Thêm chế độ Multi-tool khi UseExternalSelection = TRUE.
- Multi-tool Core chỉ tạo PCS, chạy Approach, chờ PickerSafe và thoát PCS.
- Tool DOWN/GRIP/UP do FB_ToolManager bên ngoài điều khiển.
===============================================================================
*)

//=============================================================================
// 01. CHUYỂN ĐỔI GỐC CONVEYOR SANG KIỂU POSE CỦA SOFTMOTION
//=============================================================================

// Chuyển tọa độ X của gốc conveyor.
stConveyorOriginSMC.X := ConveyorOrigin.X;
// Chuyển tọa độ Y của gốc conveyor.
stConveyorOriginSMC.Y := ConveyorOrigin.Y;
// Chuyển tọa độ Z của gốc conveyor.
stConveyorOriginSMC.Z := ConveyorOrigin.Z;
// Chuyển góc A của gốc conveyor.
stConveyorOriginSMC.A := ConveyorOrigin.A;
// Chuyển góc B của gốc conveyor.
stConveyorOriginSMC.B := 0.0;
// Chuyển góc C của gốc conveyor.
stConveyorOriginSMC.C := 0.0;

//=============================================================================
// 02. CHUYỂN ĐỔI POSE OBJECT BAN ĐẦU SANG KIỂU SOFTMOTION
//=============================================================================

// Chuyển tọa độ X của object ban đầu.
stInitialObjectSMC.X := Runtime.PCSInfo.InitialObjectPos.X;

// Chuyển tọa độ Y của object ban đầu.
stInitialObjectSMC.Y := Runtime.PCSInfo.InitialObjectPos.Y;

// Chuyển tọa độ Z của object ban đầu.
stInitialObjectSMC.Z := Runtime.PCSInfo.InitialObjectPos.Z;

// Chuyển góc A của object ban đầu.
stInitialObjectSMC.A := Runtime.PCSInfo.InitialObjectPos.A;

// // Chuyển góc B của object ban đầu.
// stInitialObjectSMC.B :=
//     REAL_TO_LREAL(Runtime.PCSInfo.InitialObjectPos.B);
// 
// // Chuyển góc C của object ban đầu.
// stInitialObjectSMC.C :=
//     REAL_TO_LREAL(Runtime.PCSInfo.InitialObjectPos.C);

//=============================================================================
// 03. GỌI MC_TrackConveyorBelt MỖI VÒNG QUÉT
//-----------------------------------------------------------------------------
// Không đặt lời gọi này chỉ trong một CASE state.
// Không hạ xTrackExecute ngay khi fbTrackBelt.Done.
//=============================================================================

fbTrackBelt(
    // Axis Group robot SCARA hiện tại.
    AxisGroup := SCARA_B,

    // Logical Axis conveyor đã chạy trong chương trình test.
    ConveyorBelt := SM_Drive_Logical_B,

    // Execute nội bộ điều khiển vòng đời PCS.
    Execute := xTrackExecute,

    // Gốc conveyor trong hệ robot/base.
    ConveyorBeltOrigin := stConveyorOriginSMC,

    // Pose object tại thời điểm tham chiếu ban đầu.
    InitialObjectPosition := stInitialObjectSMC,

    // Dùng PCS_1 cho ứng dụng Conveyor Tracking.
    CoordSystem := SMC_COORD_SYSTEM.PCS_2

);

//=============================================================================
// 04. CẬP NHẬT OUTPUT CHUNG
//=============================================================================

// Done của Manager là xung một chu kỳ.
Runtime.Response.Done := FALSE;

// SyncOK chỉ TRUE khi Robot đã tới Approach và PCS còn InUse.
SyncOK := FALSE;

// Released là xung một chu kỳ khi Multi-tool Core đã thoát PCS.
Released := FALSE;

// MotionRequest phản ánh trạng thái request nội bộ đang chờ Adapter nhận.
MotionRequest := xMotionRequestPending;

// TrackingActive TRUE khi Manager Busy, PCS Execute hoặc PCS đang InUse.
TrackingActive := Runtime.Response.Busy OR xTrackExecute OR fbTrackBelt.InUse;

// Đồng bộ trạng thái InUse của PCS vào Runtime.
Runtime.PCSInfo.InUse := fbTrackBelt.InUse;

//=============================================================================
// 05. RESET TOÀN BỘ MANAGER
//=============================================================================

IF Reset THEN
    // Đưa state machine về IDLE.
    Runtime.State := E_TrackingState.TRK_IDLE;

    // Xóa phản hồi Accepted.
    Runtime.Response.Accepted := FALSE;

    // Xóa phản hồi Busy.
    Runtime.Response.Busy := FALSE;

    // Xóa phản hồi Done.
    Runtime.Response.Done := FALSE;

    // Xóa phản hồi Error.
    Runtime.Response.Error := FALSE;

    // Xóa mã lỗi.
    Runtime.Response.ErrorID := 0;

    // Xóa index object active.
    Runtime.SelectedObjectIndex := 0;

    // Xóa ObjectID active.
    Runtime.SelectedObjectID := 0;

    // Xóa kết quả gắp.
    Runtime.PickSuccess := FALSE;

    // Đánh dấu PCS chưa hợp lệ.
    Runtime.PCSInfo.Valid := FALSE;

    // Đánh dấu PCS không còn được sử dụng.
    Runtime.PCSInfo.InUse := FALSE;

    // Hạ Execute của MC_TrackConveyorBelt.
    xTrackExecute := FALSE;

    // Xóa cờ đã phát motion.
    xMotionIssued := FALSE;

    // Xóa request motion đang chờ.
    xMotionRequestPending := FALSE;

    // Xóa trạng thái motion active.
    xMotionActive := FALSE;

    // Xóa trạng thái đã hút được vật.
    xVacuumCaptured := FALSE;

    // Tắt yêu cầu van hút.
    VacuumCommand := FALSE;

    // Tắt yêu cầu van thổi.
    BlowCommand := FALSE;

    // Hạ yêu cầu abort motion.
    MotionAbort := FALSE;

    // Xóa trạng thái đồng bộ và xung Release.
    SyncOK := FALSE;
    Released := FALSE;

    // Reset timer PickDelay.
    tonPickDelay(IN := FALSE);

    // Reset timer VacuumTimeout.
    tonVacuumTimeout(IN := FALSE);

    // Reset timer Blow.
    tonBlow(IN := FALSE);
	
	stToolSyncPos.X := 0.0;
	stToolSyncPos.Y := 0.0;
	stToolSyncPos.Z := 0.0;
	stToolSyncPos.A := 0.0;
	xPickPositionReady := FALSE;
	xPickMotionBusySeen := FALSE;
	xRetractMotionBusySeen := FALSE;
    // Kết thúc xử lý trong cycle reset.
	
	xPCSStartCaptured := FALSE;
	lrConveyorPosAtPCSStart := 0.0;
	lrDeltaCaptureToPCS := 0.0;

    RETURN;
END_IF;

//=============================================================================
// 06. HẠ EXECUTE KHI MANAGER ĐANG BUSY -> ABORT CÓ KIỂM SOÁT
//=============================================================================

//=============================================================================
// EXECUTE BỊ HẠ TRONG KHI MANAGER CHƯA KẾT THÚC
//=============================================================================
//=============================================================================
// EXECUTE ĐÃ HẠ - KHÔNG CHO STATE MACHINE TIẾP TỤC REQUEST CŨ
//=============================================================================

IF NOT Execute
AND Runtime.State <> E_TrackingState.TRK_IDLE
AND Runtime.State <> E_TrackingState.TRK_COMPLETE
AND Runtime.State <> E_TrackingState.TRK_ABORTING
AND Runtime.State <> E_TrackingState.TRK_ERROR THEN
    Runtime.State := E_TrackingState.TRK_ABORTING;
END_IF;


//=============================================================================
// 07. STATE MACHINE CHÍNH
//=============================================================================

CASE Runtime.State OF

    //=========================================================================
    // TRK_IDLE
    // Chờ lệnh Execute từ Application Manager hoặc chương trình test.
    //=========================================================================
    E_TrackingState.TRK_IDLE:

        // Manager chưa tiếp nhận lệnh.
        Runtime.Response.Accepted := FALSE;

        // Manager không bận.
        Runtime.Response.Busy := FALSE;

        // Xóa lỗi cũ khi về IDLE.
        Runtime.Response.Error := FALSE;

        // Xóa mã lỗi cũ.
        Runtime.Response.ErrorID := 0;

        // Không có object active.
        Runtime.SelectedObjectIndex := 0;

        // Không có ObjectID active.
        Runtime.SelectedObjectID := 0;

        // Xóa trạng thái gắp.
        Runtime.PickSuccess := FALSE;

        // Tắt hút.
        VacuumCommand := FALSE;

        // Tắt thổi.
        BlowCommand := FALSE;

        // Hạ abort motion.
        MotionAbort := FALSE;

        // Xóa cờ motion.
        xMotionIssued := FALSE;
        xMotionRequestPending := FALSE;
        xMotionActive := FALSE;

        // Xóa trạng thái tool đã giữ vật.
        xVacuumCaptured := FALSE;

        // Khi Execute TRUE, tiếp nhận lệnh và bắt đầu tìm object.
        IF Execute THEN
            // Báo đã tiếp nhận request.
            Runtime.Response.Accepted := TRUE;

            // Báo Manager đang bận.
            Runtime.Response.Busy := TRUE;

            // Chuyển sang Scheduler.
            Runtime.State := E_TrackingState.TRK_FIND_OBJECT;
        END_IF;

//     //=========================================================================
//     // TRK_FIND_OBJECT
//     // Scheduler tìm object phù hợp nhất trong Queue.
//     //=========================================================================
    E_TrackingState.TRK_FIND_OBJECT:

        VacuumCommand := FALSE;
        BlowCommand := FALSE;

        IF UseExternalSelection THEN
            IF ExternalObjectIndex = 0 THEN
				Runtime.Response.Error := FALSE;
				Runtime.Response.ErrorID := 0;
			
			ELSIF ExternalObjectIndex > GVL.C_MAX_TRACK_OBJECTS THEN
				Runtime.Response.Error := TRUE;
				Runtime.Response.ErrorID := 6501;
				Runtime.State := E_TrackingState.TRK_ERROR;
                
            ELSIF NOT Queue.Objects[ExternalObjectIndex].Valid THEN
                Runtime.Response.Error := TRUE;
                Runtime.Response.ErrorID := 6502;
                Runtime.State := E_TrackingState.TRK_ERROR;
            ELSE
                Runtime.SelectedObjectIndex := ExternalObjectIndex;
                Runtime.SelectedObjectID := Queue.Objects[ExternalObjectIndex].ObjectID;
                Runtime.State := E_TrackingState.TRK_RESERVE_OBJECT;
            END_IF;

        ELSIF TestFixedObjectMode THEN
            Runtime.SelectedObjectIndex := 1;
            Runtime.SelectedObjectID := 1;
            Queue.Objects[1].Valid := TRUE;
            Queue.Objects[1].ObjectID := 1;
            Queue.Objects[1].Reserved := FALSE;
            Queue.Objects[1].CanPick := TRUE;
            Queue.Objects[1].AbortRequired := FALSE;
            Queue.Objects[1].State := E_TrackingObjectState.OBJ_READY;
            Runtime.State := E_TrackingState.TRK_RESERVE_OBJECT;

        ELSE
            uiSelectedIndex := F_SelectTrackingObject(
                SelectMode := Config.SelectMode,
                SpecificID := Config.SpecificObjectID,
                DirectionSign := ConveyorConfig.DirectionSign,
                MinimumVisionScore := Config.MinimumVisionScore,
                Queue := Queue
            );

            IF uiSelectedIndex <> GVL.C_INVALID_INDEX THEN
                Runtime.SelectedObjectIndex := uiSelectedIndex;
                Runtime.SelectedObjectID := Queue.Objects[uiSelectedIndex].ObjectID;
                Runtime.State := E_TrackingState.TRK_RESERVE_OBJECT;
            END_IF;
        END_IF;


    //=========================================================================
    // TRK_RESERVE_OBJECT
    // Kiểm tra object lần cuối rồi khóa quyền sở hữu.
    //=========================================================================
    E_TrackingState.TRK_RESERVE_OBJECT:

        // Nếu index không hợp lệ thì quay lại tìm object.
        IF Runtime.SelectedObjectIndex = GVL.C_INVALID_INDEX THEN
            Runtime.State := E_TrackingState.TRK_FIND_OBJECT;

        // Nếu slot không còn hợp lệ thì hủy lựa chọn.
        ELSIF NOT Queue.Objects[Runtime.SelectedObjectIndex].Valid THEN

            Runtime.SelectedObjectIndex := 0;
            Runtime.SelectedObjectID := 0;

            Runtime.State := E_TrackingState.TRK_FIND_OBJECT;

        // Nếu object đã bị module khác Reserve thì báo lỗi tranh chấp.
        ELSIF Queue.Objects[Runtime.SelectedObjectIndex].Reserved THEN

            Runtime.Response.Error := TRUE;
            Runtime.Response.ErrorID := 6001;

            Runtime.State := E_TrackingState.TRK_ERROR;

        // Nếu object không còn đủ điều kiện gắp thì đánh dấu MISSED.
        ELSIF NOT Queue.Objects[Runtime.SelectedObjectIndex].CanPick THEN

            Queue.Objects[Runtime.SelectedObjectIndex].State := E_TrackingObjectState.OBJ_MISSED;

            // MissCode 1: mất điều kiện trước khi Reserve.
            Queue.Objects[Runtime.SelectedObjectIndex].MissCode := 1;

            Queue.Objects[Runtime.SelectedObjectIndex].Reserved := FALSE;

            Runtime.SelectedObjectIndex := 0;
            Runtime.SelectedObjectID := 0;

            Runtime.State := E_TrackingState.TRK_FIND_OBJECT;

        ELSE
            // Khóa object cho Manager này.
            Queue.Objects[Runtime.SelectedObjectIndex].Reserved := TRUE;

            // Chuyển trạng thái object sang RESERVED.
            Queue.Objects[Runtime.SelectedObjectIndex].State := E_TrackingObjectState.OBJ_RESERVED;

            // Ghi ActiveIndex vào Queue.
            Queue.ActiveIndex := Runtime.SelectedObjectIndex;

            // Xóa trạng thái hút cũ.
            xVacuumCaptured := FALSE;

            // Xóa kết quả gắp cũ.
            Runtime.PickSuccess := FALSE;

            // Chuyển sang kiểm tra vùng gắp.
            Runtime.State := E_TrackingState.TRK_WAIT_PICK_ZONE;
        END_IF;

    //=========================================================================
    // TRK_WAIT_PICK_ZONE
    // Chờ object còn nằm trong vùng an toàn và đủ thời gian.
    //=========================================================================
    E_TrackingState.TRK_WAIT_PICK_ZONE:

        // Nếu object mất hiệu lực thì giải phóng.
        IF NOT Queue.Objects[Runtime.SelectedObjectIndex].Valid THEN

            Runtime.State := E_TrackingState.TRK_RELEASE_OBJECT;

        // Nếu object đã qua mốc Abort trước khi tạo PCS.
        ELSIF Queue.Objects[Runtime.SelectedObjectIndex].AbortRequired THEN

            Queue.Objects[Runtime.SelectedObjectIndex].State := E_TrackingObjectState.OBJ_MISSED;

            // MissCode 2: quá vùng trong WAIT_PICK_ZONE.
            Queue.Objects[Runtime.SelectedObjectIndex].MissCode := 2;

            Runtime.State := E_TrackingState.TRK_RELEASE_OBJECT;

        // Nếu object còn đủ điều kiện gắp thì chuẩn bị PCS.
        ELSIF Queue.Objects[Runtime.SelectedObjectIndex].CanPick THEN

            Runtime.State := E_TrackingState.TRK_PREPARE_PCS;
        END_IF;

    //=========================================================================
    // TRK_PREPARE_PCS
    // Chụp dữ liệu object active và tạo các điểm trong PCS.
    //=========================================================================
    E_TrackingState.TRK_PREPARE_PCS:

        // Sao chép object active để tránh đọc rời rạc nhiều lần.
        stSelectedObject := Queue.Objects[Runtime.SelectedObjectIndex];

        // Lưu ObjectID vào thông tin PCS.
        Runtime.PCSInfo.ObjectID := stSelectedObject.ObjectID;

        //=========================================================================
        // CHỌN NGUỒN VỊ TRÍ OBJECT
        //-------------------------------------------------------------------------
        // Trong chế độ test:
        //     dùng vị trí object cố định.
        //
        // Trong chế độ chạy thật:
		//     dùng Pose chuẩn của Object trong Queue.
		//     Sensor/Vision đều phải chuẩn hóa về PoseInConveyor.
        //=========================================================================
        IF TestFixedObjectMode THEN
        
            // Gán vị trí object test cố định.
            Runtime.PCSInfo.InitialObjectPos.X := FixedObjectPosition.X;
        
            Runtime.PCSInfo.InitialObjectPos.Y := FixedObjectPosition.Y;
        
            Runtime.PCSInfo.InitialObjectPos.Z := FixedObjectPosition.Z;
        
            Runtime.PCSInfo.InitialObjectPos.A := FixedObjectPosition.A;
        

        
        ELSE			
			// Chế độ chạy thật lấy Pose chuẩn của Object trong hệ Conveyor.
			// Sensor/Vision đều phải chuẩn hóa dữ liệu vào PoseInConveyor
			// trước khi đưa Object vào Tracking Queue.
			
			
			Runtime.PCSInfo.InitialObjectPos := stSelectedObject.PoseInConveyor;
			
			//=============================================================
			// BÙ CHIỀU CAO MẶT HÚT SẢN PHẨM
			//=============================================================
			IF UseExternalSelection THEN
		
				Runtime.PCSInfo.InitialObjectPos.Z :=
					stSelectedObject.PoseInConveyor.Z
					+ ExternalPickSurfaceHeightMM;
		
			END_IF;
			
			
        END_IF;

        // Lưu gốc conveyor.
        //Runtime.PCSInfo.ConveyorOrigin := ConveyorOrigin;
        // Tọa độ X của gốc conveyor trong hệ robot/base.
        Runtime.PCSInfo.ConveyorOrigin.X := ConveyorOrigin.X;
        
        // Tọa độ Y của gốc conveyor trong hệ robot/base.
        Runtime.PCSInfo.ConveyorOrigin.Y := ConveyorOrigin.Y;
        
        // Tọa độ Z của gốc conveyor trong hệ robot/base.
        Runtime.PCSInfo.ConveyorOrigin.Z := ConveyorOrigin.Z;
        
        // Góc A của hệ conveyor.
        Runtime.PCSInfo.ConveyorOrigin.A := ConveyorOrigin.A;
    

        // Lưu vị trí conveyor tại thời điểm capture.
        //Runtime.PCSInfo.ConveyorCapturePos := stSelectedObject.CaptureConveyorPos;
		
		Runtime.PCSInfo.ConveyorCapturePos := LREAL_TO_REAL(stSelectedObject.CaptureConveyorPositionMM);
	
	
       // Quy ước:
		// - PickPos: điểm gắp thật của đầu Tool.
		// - ApproachPos: vị trí robot bắt đầu bám, phía trên PickPos.
		// - stToolSyncPos: cùng vị trí với ApproachPos.
		// - UseUpDown chỉ quyết định ai đi quãng cuối:
		//      TRUE  -> Tool cylinder đi xuống.
		//      FALSE -> Robot đi xuống.
		//=========================================================================
		IF UseExternalSelection THEN
		
			//---------------------------------------------------------------------
			// 1. ĐIỂM GẮP THẬT
			//---------------------------------------------------------------------
			Runtime.PickPos := ExternalPickOffset;
		
			//---------------------------------------------------------------------
			// 2. ĐIỂM ĐỒNG BỘ CỦA ROBOT
			// Luôn cao hơn điểm gắp bằng ApproachHeight,
			// không phụ thuộc Tool có Up/Down hay không.
			//---------------------------------------------------------------------
			Runtime.ApproachPos := Runtime.PickPos;
		
			Runtime.ApproachPos.Z := Runtime.PickPos.Z + ExternalApproachHeight;
		
			//---------------------------------------------------------------------
			// Robot bám conveyor tại chính điểm Approach.
			//---------------------------------------------------------------------
			stToolSyncPos := Runtime.ApproachPos;
		
			//---------------------------------------------------------------------
			// 3. ĐIỂM NÂNG SAU KHI GẮP
			// RetractHeight được tính từ điểm gắp thật.
			//---------------------------------------------------------------------
			Runtime.RetractPos := Runtime.PickPos;
		
			Runtime.RetractPos.Z := Runtime.PickPos.Z+ Config.RetractHeight;
		
		ELSE
		
			//---------------------------------------------------------------------
			// GIỮ LOGIC TRACKING THƯỜNG
			//---------------------------------------------------------------------
			Runtime.PickPos := Config.PickOffset;
		
			Runtime.ApproachPos := Config.PickOffset;
		
			Runtime.ApproachPos.Z :=
				Runtime.ApproachPos.Z
				+ Config.ApproachHeight;
		
			stToolSyncPos := Runtime.ApproachPos;
		
			Runtime.RetractPos := Config.PickOffset;
		
			Runtime.RetractPos.Z :=
				Runtime.RetractPos.Z
				+ Config.RetractHeight;
		
		END_IF;

	
		// Chu trình mới chưa tới vị trí sẵn sàng thao tác Tool.
		xPickPositionReady := FALSE;
		xPickMotionBusySeen := FALSE;
		xRetractMotionBusySeen := FALSE;
		xExitPCSTargetValid := FALSE;
        // PCS chưa hợp lệ trước khi SoftMotion báo Done.
        Runtime.PCSInfo.Valid := FALSE;
		
		// Cho phép PCS mới chụp lại Conveyor Position.
		// Mỗi Object mới vào TRK_PREPARE_PCS sẽ reset cờ này.
		xPCSStartCaptured := FALSE;

        // Chuyển sang tạo PCS.
        Runtime.State := E_TrackingState.TRK_CREATE_PCS;
		
		
	//=========================================================================
	// TRK_CREATE_PCS
	// Chốt vị trí Conveyor và tạo cạnh Execute cho MC_TrackConveyorBelt.
	//=========================================================================
	E_TrackingState.TRK_CREATE_PCS:
	
		//---------------------------------------------------------------------
		// CHỐT DỮ LIỆU PCS MỘT LẦN
		//---------------------------------------------------------------------
		IF NOT xPCSStartCaptured THEN
	
			// Vị trí Conveyor gần nhất trước lúc MC_TrackConveyorBelt Execute.
			lrConveyorPosAtPCSStart :=
				REAL_TO_LREAL(ConveyorStatus.PositionMM);
	
			// Conveyor đã dịch từ lúc Sensor/Vision Capture tới lúc tạo PCS.
			lrDeltaCaptureToPCS :=
				lrConveyorPosAtPCSStart
				- stSelectedObject.CaptureConveyorPositionMM;
	
			//-----------------------------------------------------------------
			// CẬP NHẬT POSE OBJECT TẠI THỜI ĐIỂM BẮT ĐẦU PCS
			//-----------------------------------------------------------------
			IF NOT TestFixedObjectMode THEN
	
// 				// PoseInConveyor là Pose tại thời điểm Capture.
// 				Runtime.PCSInfo.InitialObjectPos :=
// 					stSelectedObject.PoseInConveyor;
	
				// Conveyor chạy theo +X của Conveyor CS.
				Runtime.PCSInfo.InitialObjectPos.X :=
					stSelectedObject.PoseInConveyor.X
					+ LREAL_TO_REAL(lrDeltaCaptureToPCS);
	
			END_IF;
	
			// Đánh dấu đã chốt dữ liệu cho PCS hiện tại.
			xPCSStartCaptured := TRUE;
	
		END_IF;
	
		//---------------------------------------------------------------------
		// TẠO CẠNH EXECUTE CHO MC_TrackConveyorBelt
		//---------------------------------------------------------------------
		xTrackExecute := TRUE;
	
		// Sang state chờ SoftMotion tạo PCS.
		Runtime.State := E_TrackingState.TRK_WAIT_PCS;
	
	
	//=========================================================================
	// TRK_WAIT_PCS
	// Chờ MC_TrackConveyorBelt hoàn tất tạo PCS.
	//=========================================================================
	E_TrackingState.TRK_WAIT_PCS:
	
		// Quan trọng:
		// Giữ Execute TRUE trong toàn bộ vòng đời PCS.
		xTrackExecute := TRUE;
	
		//---------------------------------------------------------------------
		// TRACK CONVEYOR ERROR
		//---------------------------------------------------------------------
		IF fbTrackBelt.Error THEN
	
			Runtime.Response.Error := TRUE;
			Runtime.Response.ErrorID :=
				TO_UDINT(fbTrackBelt.ErrorID);
	
			Runtime.State :=
				E_TrackingState.TRK_ERROR;
	
		//---------------------------------------------------------------------
		// PCS ĐÃ ĐƯỢC TẠO
		//---------------------------------------------------------------------
		ELSIF fbTrackBelt.Done THEN
	
			// Không hạ xTrackExecute ở đây.
			Runtime.PCSInfo.Valid := TRUE;
	
			// Đánh dấu Object đã có Dynamic PCS.
			Queue.Objects[Runtime.SelectedObjectIndex].State :=
				E_TrackingObjectState.OBJ_PCS_READY;
	
			// Chuẩn bị phát Motion Approach.
			xMotionIssued := FALSE;
			xMotionRequestPending := FALSE;
			xMotionActive := FALSE;
	
			Runtime.State :=
				E_TrackingState.TRK_MOVE_APPROACH;
	
		END_IF;

//     //=========================================================================
//     // TRK_CREATE_PCS
//     // Tạo cạnh Execute cho MC_TrackConveyorBelt.
//     //=========================================================================
//     E_TrackingState.TRK_CREATE_PCS:
// 
//         // Bật Execute PCS.
//         xTrackExecute := TRUE;
// 
//         // Chuyển sang chờ SoftMotion tạo PCS.
//         Runtime.State := E_TrackingState.TRK_WAIT_PCS;
// 
//     //=========================================================================
//     // TRK_WAIT_PCS
//     // Chờ MC_TrackConveyorBelt hoàn tất tạo PCS.
//     //=========================================================================
//     E_TrackingState.TRK_WAIT_PCS:
// 
//         // Nếu SoftMotion báo lỗi.
//         IF fbTrackBelt.Error THEN
//             Runtime.Response.Error := TRUE;
// 
//             // Cast ErrorID theo kiểu Runtime đang sử dụng.
//             Runtime.Response.ErrorID := TO_UDINT(fbTrackBelt.ErrorID);
// 
//             Runtime.State := E_TrackingState.TRK_ERROR;
// 
//         // Khi PCS đã được tạo.
//         ELSIF fbTrackBelt.Done THEN
//             // Không hạ xTrackExecute tại đây.
//             Runtime.PCSInfo.Valid := TRUE;
// 
//             // Đánh dấu object đã có PCS.
//             Queue.Objects[Runtime.SelectedObjectIndex].State := E_TrackingObjectState.OBJ_PCS_READY;
// 
//             // Chuẩn bị phát motion Approach.
//             xMotionIssued := FALSE;
//             xMotionRequestPending := FALSE;
//             xMotionActive := FALSE;
// 
//             Runtime.State := E_TrackingState.TRK_MOVE_APPROACH;
//         END_IF;

    //=========================================================================
    // TRK_MOVE_APPROACH
    // Đi tới phía trên object trong PCS_1.
    //=========================================================================
    E_TrackingState.TRK_MOVE_APPROACH:

    // Trong chế độ test cố định, không cho Updater abort object test.
    IF TestFixedObjectMode THEN
        Queue.Objects[Runtime.SelectedObjectIndex].AbortRequired := FALSE;
    END_IF;

    // Chỉ tạo một request mới khi chưa có request/motion nào active.
    IF NOT xMotionIssued AND NOT xMotionRequestPending AND NOT xMotionActive THEN

        // Điểm đích Approach trong PCS_1.
        MotionTarget := Runtime.ApproachPos;

        // Tốc độ Approach lấy từ Tracking Config.
        MotionSpeed := Config.Motion.Approach.Speed;

        // Gia tốc Approach.
        MotionAcceleration := Config.Motion.Approach.Acceleration;

        // Giảm tốc Approach.
        MotionDeceleration := Config.Motion.Approach.Deceleration;

        // Jerk Approach.
        MotionJerk := Config.Motion.Approach.Jerk;

        // Blend radius của Approach.
        MotionBlendRadius := Config.Motion.Approach.BlendRadius;

        // Approach được thực hiện trong PCS động số 1.
        MotionCoordSystem := E_AppCoordSystem.APP_COORD_PCS2;

        // Mã lệnh MoveL.
        MotionCommand := 2;

        // Chỉ phát request nếu dữ liệu motion hợp lệ.
        IF MotionSpeed > 0.0 AND MotionAcceleration > 0.0 AND MotionDeceleration > 0.0 THEN

            // Đánh dấu request đang chờ Motion Adapter nhận.
            xMotionRequestPending := TRUE;

            // Đánh dấu state đã tạo request.
            xMotionIssued := TRUE;

        ELSE
            // Thông số Dynamic bằng 0 nên không được phát motion.
            Runtime.Response.Error := TRUE;

            // Mã lỗi nội bộ: cấu hình Approach không hợp lệ.
            Runtime.Response.ErrorID := 6101;

            // Chuyển sang state lỗi.
            Runtime.State := E_TrackingState.TRK_ERROR;
        END_IF;
    END_IF;

    // Motion Adapter đã nhận request.
    IF MotionAccepted AND xMotionRequestPending THEN

        // Hạ request pending.
        xMotionRequestPending := FALSE;

        // Bắt đầu chờ MotionDone.
        xMotionActive := TRUE;
    END_IF;

    // Motion Approach hoàn thành.
    IF MotionDone AND xMotionActive THEN
		xMotionActive := FALSE;
		xMotionIssued := FALSE;
		xMotionRequestPending := FALSE;
	
		IF UseExternalSelection THEN
			IF ExternalUseUpDown THEN
				// Robot đã tới SyncPos.
				// Tool cơ khí sẽ thực hiện hành trình xuống.
				xPickPositionReady := TRUE;
			ELSE
				// Robot mới chỉ tới SyncPos.
				// Bắt buộc phải phát thêm MoveL xuống PickPos.
				xPickPositionReady := FALSE;
			END_IF;
		ELSE
			xPickPositionReady := FALSE;
		END_IF;
	
		Runtime.State := E_TrackingState.TRK_MOVE_PICK;
	
	ELSIF MotionError AND xMotionActive THEN
		xMotionActive := FALSE;
		xMotionIssued := FALSE;
		xMotionRequestPending := FALSE;
	
		Runtime.Response.Error := TRUE;
		Runtime.Response.ErrorID := MotionErrorID;
		Runtime.State := E_TrackingState.TRK_ERROR;
	END_IF;

    //=========================================================================
    // TRK_MOVE_PICK
    // Hạ TCP từ Approach xuống PickPos trong PCS_1.
    //=========================================================================
    E_TrackingState.TRK_MOVE_PICK:

        IF UseExternalSelection THEN
            xTrackExecute := TRUE;
			VacuumCommand := FALSE;
			BlowCommand := FALSE;
	
			//---------------------------------------------------------------------
			// Chưa tới vị trí sẵn sàng thì phát một MoveL trong PCS_1.
			//---------------------------------------------------------------------
			IF NOT xPickPositionReady THEN

				IF NOT xMotionIssued AND NOT xMotionRequestPending AND NOT xMotionActive THEN
			
					Queue.Objects[Runtime.SelectedObjectIndex].State := E_TrackingObjectState.OBJ_PICKING;
			
					// Không có Up/Down:
					// robot phải tự xuống điểm Pick thật.
					MotionTarget := Runtime.PickPos;
			
					MotionSpeed := Config.Motion.Pick.Speed;
					MotionAcceleration := Config.Motion.Pick.Acceleration;
					MotionDeceleration := Config.Motion.Pick.Deceleration;
					MotionJerk := Config.Motion.Pick.Jerk;
					MotionBlendRadius := Config.Motion.Pick.BlendRadius;
					MotionCoordSystem := E_AppCoordSystem.APP_COORD_PCS2;
					MotionCommand := 2;
			
					xPickMotionBusySeen := FALSE;
					xMotionRequestPending := TRUE;
					xMotionIssued := TRUE;
				END_IF;
			
				IF MotionAccepted AND xMotionRequestPending THEN
					xMotionRequestPending := FALSE;
					xMotionActive := TRUE;
				END_IF;
			
				IF xMotionActive AND MotionBusy THEN
					xPickMotionBusySeen := TRUE;
				END_IF;
			
				IF MotionDone
				AND xMotionActive
				AND xPickMotionBusySeen THEN
			
					xMotionActive := FALSE;
					xMotionIssued := FALSE;
					xMotionRequestPending := FALSE;
					xPickMotionBusySeen := FALSE;
			
					// Chỉ tới đây mới xác nhận robot đã xuống PickPos.
					xPickPositionReady := TRUE;
			
				ELSIF MotionError AND xMotionActive THEN
			
					xMotionActive := FALSE;
					xMotionIssued := FALSE;
					xMotionRequestPending := FALSE;
					xPickMotionBusySeen := FALSE;
			
					Runtime.Response.Error := TRUE;
					Runtime.Response.ErrorID := MotionErrorID;
					Runtime.State := E_TrackingState.TRK_ERROR;
				END_IF;
			
			END_IF;
	
			//---------------------------------------------------------------------
			// Chỉ báo SyncOK sau khi robot tới đúng vị trí thao tác.
			//---------------------------------------------------------------------
			SyncOK := xPickPositionReady AND Runtime.PCSInfo.Valid AND fbTrackBelt.InUse;
	
			//---------------------------------------------------------------------
			// Controller đã hoàn thành:
			// - Có Up/Down: DOWN -> GRIP -> UP.
			// - Không Up/Down: GRIP.
			//---------------------------------------------------------------------
			IF PickerSafe AND SyncOK THEN
	
				Runtime.PickSuccess := TRUE;
				xVacuumCaptured := TRUE;
				
				xRetractMotionBusySeen := FALSE;
				xExitPCSTargetValid := FALSE;
				
				IF ExternalUseUpDown THEN
					// Tool đã thực hiện DOWN -> GRIP -> UP.
					// Robot vẫn đang tại Sync/ApproachPos.
					// Không được chạy xuống RetractPos.
					Runtime.State := E_TrackingState.TRK_LEAVE_PCS;
				ELSE
					// Không có Tool Up/Down.
					// Robot đang tại PickPos và cần tự nâng lên RetractPos.
					Runtime.State := E_TrackingState.TRK_MOVE_RETRACT;
				END_IF;
					
			ELSIF fbTrackBelt.Error THEN
	
				Runtime.Response.Error := TRUE;
				Runtime.Response.ErrorID :=
					TO_UDINT(fbTrackBelt.ErrorID);
				Runtime.State := E_TrackingState.TRK_ERROR;
	
			END_IF;

        ELSE


            // Chưa VacuumOK nên vẫn có thể abort nếu object quá vùng.
            IF Queue.Objects[Runtime.SelectedObjectIndex].AbortRequired AND NOT xVacuumCaptured THEN

                Queue.Objects[Runtime.SelectedObjectIndex].State := E_TrackingObjectState.OBJ_MISSED;

                // MissCode 4: quá vùng trong Move Pick.
                Queue.Objects[Runtime.SelectedObjectIndex].MissCode := 4;

                MotionAbort := TRUE;

                Runtime.State := E_TrackingState.TRK_ABORT_ACTIVE;

            ELSE
                // Tạo request Pick mới.
                IF NOT xMotionIssued AND NOT xMotionRequestPending AND NOT xMotionActive THEN

                    // Đánh dấu object đang ở pha Picking.
                    Queue.Objects[Runtime.SelectedObjectIndex].State := E_TrackingObjectState.OBJ_PICKING;

                    // Gán điểm Pick.
                    MotionTarget := Runtime.PickPos;

                    // Gán tốc độ Pick.
                    MotionSpeed := Config.Motion.Pick.Speed;

                    // Gán gia tốc Pick.
                    MotionAcceleration := Config.Motion.Pick.Acceleration;

                    // Gán giảm tốc Pick.
                    MotionDeceleration := Config.Motion.Pick.Deceleration;

                    // Gán jerk Pick.
                    MotionJerk := Config.Motion.Pick.Jerk;

                    // Gán blend Pick.
                    MotionBlendRadius := Config.Motion.Pick.BlendRadius;

                    // Pick chạy trong PCS_1.
                    MotionCoordSystem := E_AppCoordSystem.APP_COORD_PCS2;

                    // Mã lệnh MoveL.
                    MotionCommand := 2;

                    // Bật request pending.
                    xMotionRequestPending := TRUE;

                    // Đánh dấu đã tạo lệnh.
                    xMotionIssued := TRUE;
                END_IF;
					
					// Adapter đã nhận đúng request Pick.
					IF MotionAccepted AND xMotionRequestPending THEN
						xMotionRequestPending := FALSE;
						xMotionActive := TRUE;
					END_IF;
					
					// Phải thấy motion Pick thực sự Busy ít nhất một scan.
					// Nhờ đó không nhận nhầm Done còn lại từ lệnh Approach.
					IF xMotionActive AND MotionBusy THEN
						xPickMotionBusySeen := TRUE;
					END_IF;
					
					// Chỉ công nhận Done sau khi motion Pick đã thực sự Busy.
					IF MotionDone
					AND xMotionActive
					AND xPickMotionBusySeen THEN
					
						xMotionActive := FALSE;
						xMotionIssued := FALSE;
						xMotionRequestPending := FALSE;
						xPickMotionBusySeen := FALSE;
					
						xPickPositionReady := TRUE;
					
					ELSIF MotionError AND xMotionActive THEN
					
						xMotionActive := FALSE;
						xMotionIssued := FALSE;
						xMotionRequestPending := FALSE;
						xPickMotionBusySeen := FALSE;
					
						Runtime.Response.Error := TRUE;
						Runtime.Response.ErrorID := MotionErrorID;
						Runtime.State := E_TrackingState.TRK_ERROR;
					
					END_IF;

//                 // Adapter đã nhận request.
//                 IF MotionAccepted AND xMotionRequestPending THEN
//                     xMotionRequestPending := FALSE;
//                     xMotionActive := TRUE;
//                 END_IF;
// 
//                 // Motion Pick hoàn thành.
//                 IF MotionDone AND xMotionActive THEN
//                     xMotionActive := FALSE;
//                     xMotionIssued := FALSE;
// 
//                     Runtime.State := E_TrackingState.TRK_GRIP_ON;
// 
//                 // Motion Pick lỗi.
//                 ELSIF MotionError AND xMotionActive THEN
//                     xMotionActive := FALSE;
// 
//                     Runtime.Response.Error := TRUE;
//                     Runtime.Response.ErrorID := MotionErrorID;
// 
//                     Runtime.State := E_TrackingState.TRK_ERROR;
//                 END_IF;
            END_IF;

        END_IF;


    //=========================================================================
    // TRK_GRIP_ON
    // Bật hút và chờ PickDelay.
    //=========================================================================
    E_TrackingState.TRK_GRIP_ON:

        // Bật yêu cầu hút.
        VacuumCommand := TRUE;

        // Chạy timer PickDelay.
        tonPickDelay(
            IN := TRUE,
            PT := Config.PickDelay
        );

        // Khi hết thời gian chờ.
        IF tonPickDelay.Q THEN
            // Reset timer PickDelay.
            tonPickDelay(IN := FALSE);

            // Reset timer VacuumTimeout.
            tonVacuumTimeout(IN := FALSE);

            // Chuyển sang chờ VacuumOK.
            Runtime.State := E_TrackingState.TRK_WAIT_GRIP;
        END_IF;

    //=========================================================================
    // TRK_WAIT_GRIP
    // Chờ VacuumOK hoặc timeout.
    //=========================================================================
    E_TrackingState.TRK_WAIT_GRIP:

        // Giữ hút trong toàn bộ thời gian chờ.
        VacuumCommand := TRUE;

        // Chạy timer VacuumTimeout.
        tonVacuumTimeout(
            IN := TRUE,
            PT := Config.VacuumTimeout
        );

        // Nếu tool đã giữ được vật.
        IF VacuumOK THEN
            // Reset timeout.
            tonVacuumTimeout(IN := FALSE);

            // Khóa trạng thái đã hút thành công.
            xVacuumCaptured := TRUE;

            // Báo gắp thành công.
            Runtime.PickSuccess := TRUE;

            // Chuẩn bị phát motion Retract.
            xMotionIssued := FALSE;
            xMotionRequestPending := FALSE;
            xMotionActive := FALSE;

            Runtime.State := E_TrackingState.TRK_MOVE_RETRACT;

        // Nếu hết timeout mà chưa hút được.
        ELSIF tonVacuumTimeout.Q THEN
            // Reset timer.
            tonVacuumTimeout(IN := FALSE);

            // Tăng số lần thử.
            Queue.Objects[Runtime.SelectedObjectIndex].PickAttempts := Queue.Objects[Runtime.SelectedObjectIndex].PickAttempts + 1;

            // Nếu object đã vượt vùng an toàn thì không thử lại.
            IF Queue.Objects[Runtime.SelectedObjectIndex].AbortRequired THEN

                VacuumCommand := FALSE;

                Queue.Objects[Runtime.SelectedObjectIndex].State := E_TrackingObjectState.OBJ_MISSED;

                // MissCode 5: timeout và đã vượt vùng.
                Queue.Objects[Runtime.SelectedObjectIndex].MissCode := 5;

                Runtime.State := E_TrackingState.TRK_ABORT_ACTIVE;

            // Nếu còn lượt thử.
            ELSIF Queue.Objects[Runtime.SelectedObjectIndex].PickAttempts < Config.MaxPickAttempts THEN

                // Tắt hút trước lần thử tiếp theo.
                VacuumCommand := FALSE;

                // Cho phép phát lại lệnh Pick.
                xMotionIssued := FALSE;
                xMotionRequestPending := FALSE;
                xMotionActive := FALSE;

                Runtime.State := E_TrackingState.TRK_MOVE_PICK;

            ELSE
                // Hết số lần thử.
                VacuumCommand := FALSE;

                Queue.Objects[Runtime.SelectedObjectIndex].State := E_TrackingObjectState.OBJ_MISSED;

                // MissCode 6: hết số lần thử hút.
                Queue.Objects[Runtime.SelectedObjectIndex].MissCode := 6;

                Runtime.State := E_TrackingState.TRK_ABORT_ACTIVE;
            END_IF;
        END_IF;

    //=========================================================================
	// TRK_MOVE_RETRACT
	// Nâng sản phẩm trong PCS_1.
	//=========================================================================
	E_TrackingState.TRK_MOVE_RETRACT:
	
		// Giữ sản phẩm trong khi nâng.
		VacuumCommand := xVacuumCaptured;
		xTrackExecute := TRUE;
	
		//---------------------------------------------------------------------
		// PHÁT LỆNH RETRACT MỘT LẦN
		//---------------------------------------------------------------------
		IF NOT xMotionIssued
		AND NOT xMotionRequestPending
		AND NOT xMotionActive THEN
	
			// X/Y/A giữ nguyên theo PickPos; chỉ Z tăng.
			MotionTarget := Runtime.RetractPos;
	
			MotionSpeed := Config.Motion.Retract.Speed;
			MotionAcceleration := Config.Motion.Retract.Acceleration;
			MotionDeceleration := Config.Motion.Retract.Deceleration;
			MotionJerk := Config.Motion.Retract.Jerk;
			MotionBlendRadius := 0.0;
	
			// Vẫn bám vật trong lúc nâng.
			MotionCoordSystem := E_AppCoordSystem.APP_COORD_PCS2;
			MotionCommand := 2;
	
			xRetractMotionBusySeen := FALSE;
			xMotionRequestPending := TRUE;
			xMotionIssued := TRUE;
		END_IF;
	
		//---------------------------------------------------------------------
		// ADAPTER ĐÃ NHẬN LỆNH RETRACT
		//---------------------------------------------------------------------
		IF MotionAccepted AND xMotionRequestPending THEN
			xMotionRequestPending := FALSE;
			xMotionActive := TRUE;
		END_IF;
	
		//---------------------------------------------------------------------
		// CHÍNH LỆNH RETRACT ĐÃ THỰC SỰ CHẠY
		//---------------------------------------------------------------------
		IF xMotionActive AND MotionBusy THEN
			xRetractMotionBusySeen := TRUE;
		END_IF;
	
		//---------------------------------------------------------------------
		// RETRACT HOÀN THÀNH THẬT
		//---------------------------------------------------------------------
		IF MotionDone
		AND xMotionActive
		AND xRetractMotionBusySeen THEN
	
			xMotionActive := FALSE;
			xMotionIssued := FALSE;
			xMotionRequestPending := FALSE;
			xRetractMotionBusySeen := FALSE;
		
			xExitPCSTargetValid := FALSE;
		
			Runtime.State := E_TrackingState.TRK_LEAVE_PCS;
// 			xMotionActive := FALSE;
// 			xMotionIssued := FALSE;
// 			xMotionRequestPending := FALSE;
// 			xRetractMotionBusySeen := FALSE;
// 	
// 			xExitPCSTargetValid := FALSE;
// 	
// 			//-----------------------------------------------------------------
// 			// Chỉ sau khi nâng xong mới chụp vị trí MCS hiện tại.
// 			//-----------------------------------------------------------------
// 			stExitPCSTarget.X :=
// 				TO_REAL(POU_MONITOR_ROBOT.RB1_POS.c.X);
// 	
// 			stExitPCSTarget.Y :=
// 				TO_REAL(POU_MONITOR_ROBOT.RB1_POS.c.Y);
// 	
// 			stExitPCSTarget.Z :=
// 				TO_REAL(POU_MONITOR_ROBOT.RB1_POS.c.Z);
// 	
// 			stExitPCSTarget.A :=
// 				TO_REAL(POU_MONITOR_ROBOT.RB1_POS.c.A);
// 	
// 			// Chỉ cộng thêm Z, không thay đổi X/Y/A.
// 			stExitPCSTarget.Z :=
// 				stExitPCSTarget.Z + rExitPCSOffsetZ;
// 	
// 			IF stExitPCSTarget.Z < 0.0
// 			OR stExitPCSTarget.Z > rExitPCSMaxZ THEN
// 	
// 				Runtime.Response.Error := TRUE;
// 				Runtime.Response.ErrorID := 6130;
// 				Runtime.State := E_TrackingState.TRK_ERROR;
// 	
// 			ELSE
// 	
// 				xExitPCSTargetValid := TRUE;
// 				Runtime.State := E_TrackingState.TRK_LEAVE_PCS;
// 	
// 			END_IF;
	
		ELSIF MotionError AND xMotionActive THEN
	
			xMotionActive := FALSE;
			xMotionIssued := FALSE;
			xMotionRequestPending := FALSE;
			xRetractMotionBusySeen := FALSE;
	
			Runtime.Response.Error := TRUE;
			Runtime.Response.ErrorID := MotionErrorID;
			Runtime.State := E_TrackingState.TRK_ERROR;
	
		END_IF;


	//=============================================================================
	// TRK_LEAVE_PCS — STATE 120
	//-----------------------------------------------------------------------------
	// Phát một motion ngắn trong Robot Base/MCS để AxisGroup rời PCS_1.
	//
	// stExitPCSTarget đã được chụp một lần tại cuối Retract.
	// Không cập nhật stExitPCSTarget trong state này.
	//=============================================================================
	E_TrackingState.TRK_LEAVE_PCS:
	
		// Tiếp tục giữ sản phẩm.
		VacuumCommand := xVacuumCaptured;
	
		// Giữ MC_TrackConveyorBelt hoạt động cho tới khi AxisGroup rời PCS.
		xTrackExecute := TRUE;
	
		//---------------------------------------------------------------------
		// CHỤP TARGET MCS VÀ PHÁT MOTION EXIT PCS MỘT LẦN
		//---------------------------------------------------------------------
		IF NOT xMotionIssued
		AND NOT xMotionRequestPending
		AND NOT xMotionActive THEN
	
			// Chụp vị trí MCS muộn nhất có thể,
			// ngay trước khi tạo request Motion Queue.
// 			stExitPCSTarget.X :=
// 				TO_REAL(POU_MONITOR_ROBOT.RB1_POS.c.X);
// 	
// 			stExitPCSTarget.Y :=
// 				TO_REAL(POU_MONITOR_ROBOT.RB1_POS.c.Y);
// 	
// 			stExitPCSTarget.Z :=
// 				TO_REAL(POU_MONITOR_ROBOT.RB1_POS.c.Z);
// 	
// 			stExitPCSTarget.A :=
// 				TO_REAL(POU_MONITOR_ROBOT.RB1_POS.c.A);
				
			stExitPCSTarget.X :=
				TO_REAL(POU_COORDINATE_.Pos_Out_B_MCS.c.X);
	
			stExitPCSTarget.Y :=
				TO_REAL(POU_COORDINATE_.Pos_Out_B_MCS.c.Y);
	
			stExitPCSTarget.Z :=
				TO_REAL(POU_COORDINATE_.Pos_Out_B_MCS.c.Z);
	
			stExitPCSTarget.A :=
				TO_REAL(POU_COORDINATE_.Pos_Out_B_MCS.c.A);
	
			// Chỉ nâng thêm Z; không cộng offset X/Y/A.
			stExitPCSTarget.X := stExitPCSTarget.X - rExitPCSOffsetX;
			stExitPCSTarget.Z := stExitPCSTarget.Z + rExitPCSOffsetZ;
	
			//-----------------------------------------------------------------
			// KIỂM TRA TARGET
			//-----------------------------------------------------------------
			IF stExitPCSTarget.Z < 0.0
			OR stExitPCSTarget.Z > rExitPCSMaxZ THEN
	
				Runtime.Response.Error := TRUE;
				Runtime.Response.ErrorID := 6130;
				Runtime.State := E_TrackingState.TRK_ERROR;
	
			ELSE
	
				xExitPCSTargetValid := TRUE;
	
				MotionTarget := stExitPCSTarget;
	
				MotionSpeed := 80.0;
				MotionAcceleration := 300.0;
				MotionDeceleration := 300.0;
				MotionJerk := 1000.0;
				MotionBlendRadius := 0.0;
	
				// Chạy trong Robot Base/MCS để thoát khỏi PCS_1.
				MotionCoordSystem :=
					E_AppCoordSystem.APP_COORD_ROBOT_BASE;
	
				MotionCommand := 2;
	
				xMotionRequestPending := TRUE;
				xMotionIssued := TRUE;
	
			END_IF;
	
		END_IF;
	
		//---------------------------------------------------------------------
		// ADAPTER ĐÃ NHẬN MOTION EXIT PCS
		//---------------------------------------------------------------------
		IF MotionAccepted AND xMotionRequestPending THEN
			xMotionRequestPending := FALSE;
			xMotionActive := TRUE;
		END_IF;
	
		//---------------------------------------------------------------------
		// EXIT PCS HOÀN THÀNH
		//---------------------------------------------------------------------
		IF MotionDone AND xMotionActive THEN
	
			xMotionActive := FALSE;
			xMotionIssued := FALSE;
			xMotionRequestPending := FALSE;
	
			Runtime.State := E_TrackingState.TRK_RELEASE_PCS;
	
		ELSIF MotionError AND xMotionActive THEN
	
			xMotionActive := FALSE;
			xMotionIssued := FALSE;
			xMotionRequestPending := FALSE;
	
			Runtime.Response.Error := TRUE;
			Runtime.Response.ErrorID := MotionErrorID;
			Runtime.State := E_TrackingState.TRK_ERROR;
	
		END_IF;


	//=============================================================================
	// TRK_RELEASE_PCS — STATE 130
	//-----------------------------------------------------------------------------
	// Motion Exit PCS trong MCS đã hoàn thành.
	// Chờ SoftMotion xác nhận PCS_1 không còn được AxisGroup sử dụng.
	//=============================================================================
	E_TrackingState.TRK_RELEASE_PCS:
	
		// Tiếp tục giữ sản phẩm.
		VacuumCommand := xVacuumCaptured;
	
		// Không còn motion pending.
		xMotionIssued := FALSE;
		xMotionRequestPending := FALSE;
		xMotionActive := FALSE;
	
		// Trong lúc InUse vẫn TRUE, giữ FB Track còn Execute.
		xTrackExecute := TRUE;
	
		//---------------------------------------------------------------------
		// AXIS GROUP ĐÃ RỜI PCS_1
		//---------------------------------------------------------------------
		IF NOT fbTrackBelt.InUse THEN
	
			// Bây giờ mới được hạ Execute của MC_TrackConveyorBelt.
			xTrackExecute := FALSE;
	
			Runtime.PCSInfo.Valid := FALSE;
			Runtime.PCSInfo.InUse := FALSE;
	
			xExitPCSTargetValid := FALSE;
	
			IF UseExternalSelection THEN
                Released := TRUE;
                Runtime.Response.Done := TRUE;
                Runtime.Response.Busy := FALSE;
                Runtime.State := E_TrackingState.TRK_COMPLETE;
            ELSE
                Runtime.State := E_TrackingState.TRK_MOVE_SAFE_LEAVE;
            END_IF;
	
		//---------------------------------------------------------------------
		// TRACK CONVEYOR BÁO LỖI
		//---------------------------------------------------------------------
		ELSIF fbTrackBelt.Error THEN
	
			Runtime.Response.Error := TRUE;
			Runtime.Response.ErrorID := fbTrackBelt.ErrorID;
			Runtime.State := E_TrackingState.TRK_ERROR;
		END_IF;
	
	//=============================================================================
	// TRK_MOVE_SAFE_LEAVE
	//-----------------------------------------------------------------------------
	// PCS đã được release hoàn toàn.
	// Robot thực hiện MoveL tới điểm an toàn tuyệt đối trong Robot Base.
	//
	// Config.LeavePos phải là một điểm đã được dạy và test bằng Jog/MoveL riêng.
	// Không tính bằng cách cộng offset từ TCP hiện tại.
	//=============================================================================
	E_TrackingState.TRK_MOVE_SAFE_LEAVE:
	
		// Tiếp tục giữ sản phẩm.
		VacuumCommand := xVacuumCaptured;
	
		// Không cho MC_TrackConveyorBelt hoạt động lại.
		xTrackExecute := FALSE;
	
		// Tạo request motion một lần.
		IF NOT xMotionIssued
		AND NOT xMotionRequestPending
		AND NOT xMotionActive THEN
	
			// Điểm an toàn tuyệt đối trong Robot Base.
			MotionTarget := Config.LeavePos;
	
			// Thông số chuyển động Leave.
			MotionSpeed := Config.Motion.Leave.Speed;
			MotionAcceleration := Config.Motion.Leave.Acceleration;
			MotionDeceleration := Config.Motion.Leave.Deceleration;
			MotionJerk := Config.Motion.Leave.Jerk;
	
